(* Logix 5000 project; controller VET 1756-L62 rev 19.52; software revision 19.01; part 2 of 27 *)

        [110].S.BITS1.29   // 70-CAN-12 Falla Abrir
        [129].S.BITS1.30   // RIB-30 Falla Partida
        [129].S.BITS2.11   // RED-636-00 Enc Ext
        [36].S.BITS1.10   // 7-BIN-1060 LH
        [372].S.BITS1.8   // 110-ACD-001/1 Atollo
        [36].S.BITS1.26   // 60-VEN-002 FLL
        [119].S.BITS1.2   // 70-TDC-005 Conf. Marcha
        [141].S.BITS2.20   // 7-ROS-1140 Reset Falla
        [36].S.BITS1.27   // 60-VEN-002 FV0
        [373].S.BITS1.8   // 110-EXP-001/1 Atollo
        [46].S.BITS1.30   // 7-ROS-1069 Falla Partida
        [46].S.BITS2.7   // CON-666-00 Disable Codes
        [36].S.BITS1.28   // 60-VEN-002 FATO
        [133].S.BITS1.0   // RIB-32 Enable
        [374].S.BITS1.8   // 110-DES-001/1 Atollo
        [36].S.BITS2.7   // CON-660-00Cmd Open
        [375].S.BITS1.8   // 110-CAE-001/1 Atollo
        [141].S.BITS2.23   // 7-ROS-1140 Test
        [36].S.BITS2.20   // 60-VEN-002 Reset Falla
        [235].S.BITS1.9   // Nivel lleno Estanque Faenadora
        [36].S.BITS2.23   // 60-VEN-002 Test
        [47].S.BITS1.1   // 7-ELV-1070 Falla Resumen
        [141].S.BITS2.27   // 7-ROS-1140 Cmd. Marcha
        [47].S.BITS2.7   // CON-667-00 Disable Codes
        [129].S.BITS2.20   // RIB-30 Reset Falla
        [36].S.BITS2.27   // 60-VEN-002 Cmd. Marcha
        [141].S.BITS2.30   // 7-ROS-1140 OUT MARCHA
        [131].S.BITS1.9   // 100-TDC-001 Sobrecarga
        [48].S.BITS2.7   // CON-668-00 Disable Codes
        [110].S.BITS2.31   // 70-CAN-12 OUT OPEN
        [142].S.BITS1.7   // 70-BIN-002 LLL
        [111].S.BITS1.0   // CV-5 Enable
        [111].S.BITS1.1   // CV-5 Falla Resumen
        [87].S.BITS1.0   // TCS-28 Enable
        [46].S.BITS1.10   // 90-MMA-001 Velocidad Cero
        [87].S.BITS1.1   // TCS-28 Falla Resumen
        [156].S.BITS1.9   // 7-BIN-1155 LM
        [49].S.BITS1.10   // 90-TOR-001 Velocidad Cero
        [50].S.BITS1.8   // 90-TAB-002 Atollo
        [202].S.BITS2.11   // RED-037-00 Enc Ext
        [50].S.BITS1.10   // 90-TAB-002 Velocidad Cero
        [66].S.BITS1.4   // 60-ELV-003 Cmd. Automatico
        [442].S.BITS1.8   // 9-BIN-704 LL
        [84].S.BITS1.8   // 90-MRO-003-B Atollo
        [111].S.BITS1.2   // CV-5 Conf Pos Abrir
        [684].S.BITS2.23   // 120-CAN-070 Test
        [160].S.BITS2.27   // ROS-015-00 Cmd
        [23].S.BITS1.10   // 90-CAN-010 Conf. Abierto
        [160].S.BITS2.31   // ROS-015-00 Out
        [111].S.BITS1.4   // CV-5 Conf Pos Cerrar
        [37].S.BITS1.0   // 60-VEN-004A Enable
        [444].S.BITS1.8   // 9-BIN-706 LL
        [37].S.BITS1.26   // 60-VEN-004A FLL
        [107].S.BITS1.10   // 7-BIN-1106 LH
        [156].S.BITS1.10   // 7-BIN-1155 LH
        [37].S.BITS1.27   // 60-VEN-004A FV0
        [683].S.BITS1.8   // 120-BIN-032 LL
        [25].S.BITS1.0   // 7-CON-1025 Enable
        [143].S.BITS1.26   // 7-BBA-1142 FLL
        [156].S.BITS1.29   // M1-COMP-400 Falla Abrir
        [143].S.BITS1.27   // 7-BBA-1142 FV0
        [143].S.BITS1.28   // 7-BBA-1142 FATO
        [166].S.BITS1.2   // ROS-018-00 Run
        [49].S.BITS1.30   // 7-CON-1072 Falla Cerrar
        [683].S.BITS1.9   // 120-BIN-032 LM
        [95].S.BITS1.4   // CV-7 Conf Pos Cerrar
        [143].S.BITS1.30   // 7-BBA-1142 Falla Partida
        [95].S.BITS1.8   // 7-RED-770 LL
        [111].S.BITS1.26   // RIB-21 FLL
        [111].S.BITS1.27   // RIB-21 FV0
        [143].S.BITS2.7   // CON-684-00Cmd Open
        [95].S.BITS1.10   // 7-RED-770 LH
        [111].S.BITS1.28   // RIB-21 FATO
        [44].S.BITS1.10   // 7-TV-107X LH
        [111].S.BITS1.29   // CV-5 Falla Abrir
        [449].S.BITS1.8   // 110-VAL-001/2-1 Atollo
        [111].S.BITS1.30   // CV-5 Falla Cerrar
        [54].S.BITS1.8   // 90-ALI-002 Atollo
        [111].S.BITS2.20   // CV-5 Reset Falla
        [37].S.BITS1.28   // 60-VEN-004A FATO
        [129].S.BITS2.23   // RIB-30 Test
        [147].S.BITS1.30   // 7-CON-1146 Falla Cerrar
        [299].S.BITS1.8   // 100-TDP-006 Atollo
        [111].S.BITS2.23   // CV-5 Test
        [95].S.BITS1.26   // RIB-13 FLL
        [37].S.BITS2.7   // CON-661-00Cmd Open
        [111].S.BITS2.27   // CV-5 Cmd. Open
        [37].S.BITS2.23   // 60-VEN-004A Test
        [111].S.BITS2.30   // CV-5 OUT CLOSE
        [173].S.BITS1.28   // 70-TOR-017 FATO
        [173].S.BITS1.30   // 70-TOR-017 Falla Partida
        [173].S.BITS2.20   // 70-TOR-017 Reset Falla
        [173].S.BITS2.23   // 70-TOR-017 Test
        [173].S.BITS2.27   // 70-TOR-017 Cmd. Marcha
        [38].S.BITS1.0   // 60-TOR-002Enable
        [111].S.BITS2.31   // CV-5 OUT OPEN
        [173].S.BITS2.30   // 70-TOR-017 OUT MARCHA
        [38].S.BITS1.1   // 60-TOR-002Falla Resumen
        [143].S.BITS2.30   // 7-BBA-1142 OUT MARCHA
        [174].S.BITS1.2   // ROS-022-00 Run
        [38].S.BITS1.7   // 60-tol LLL
        [129].S.BITS2.27   // RIB-30 Cmd. Marcha
        [161].S.BITS1.0   // 7-ROS-1160 Enable
        [147].S.BITS2.7   // CON-639-00 Disable Codes
        [49].S.BITS2.7   // CON-669-00 Disable Codes
        [451].S.BITS1.8   // 110-ENF-001/2-5 Atollo
        [174].S.BITS1.7   // 70-BIN-018 LLL
        [134].S.BITS1.9   // 7-TOL-1137 LM
        [38].S.BITS1.26   // 60-TOR-002FLL
        [104].S.BITS1.9   // 90-TDC-003 Sobrecarga
        [38].S.BITS1.27   // 60-TOR-002FV0
        [55].S.BITS1.10   // 90-FIL-002 Conf. Abierto
        [142].S.BITS1.9   // 100-TDC-003 Sobrecarga
        [38].S.BITS1.28   // 60-TOR-002FATO
        [170].S.BITS1.0   // Enable
        [185].S.BITS1.9   // TOL-025-00 LM
        [87].S.BITS1.2   // TCS-28 Conf. Marcha
        [95].S.BITS1.27   // RIB-13 FV0
        [171].S.BITS2.27   // 7-VRT-1169 Cmd. Marcha
        [50].S.BITS1.30   // 7-CON-1073 Falla Cerrar
        [166].S.BITS1.7   // 70-BIN-014 LLL
        [119].S.BITS1.4   // 70-TDC-005 Cmd. Automatico
        [87].S.BITS1.4   // TCS-28 Cmd. Automatico
        [87].S.BITS1.8   // ROS-615-00 IAto
        [171].S.BITS2.30   // 7-VRT-1169 OUT MARCHA
        [70].S.BITS1.8   // 70-TOL-001 LL
        [95].S.BITS1.28   // RIB-13 FATO
        [144].S.BITS1.7   // 70-BIN-003 LLL
        [56].S.BITS1.8   // 90-VEN-002 Atollo
        [38].S.BITS2.7   // CON-662-00Cmd Open
        [194].S.BITS1.7   // 70-TOL-006 LLL
        [119].S.BITS1.26   // 70-TDC-005 FLL
        [95].S.BITS1.29   // CV-7 Falla Abrir
        [119].S.BITS1.27   // 70-TDC-005 FV0
        [462].S.BITS1.8   // 9-BIN-724 LL
        [174].S.BITS2.11   // ROS-022-00 Enc Ext
        [174].S.BITS2.27   // ROS-022-00 Cmd
        [174].S.BITS2.31   // ROS-022-00 Out
        [38].S.BITS2.20   // 60-TOR-002Reset Falla
        [119].S.BITS1.28   // 70-TDC-005 FATO
        [97].S.BITS1.10   // 7-TOL-799 LH
        [170].S.BITS1.1   // Falla Resumen
        [464].S.BITS1.8   // 9-BIN-726 LL
        [54].S.BITS1.10   // 90-ALI-002 Velocidad Cero
        [95].S.BITS1.30   // CV-7 Falla Cerrar
        [38].S.BITS2.23   // 60-TOR-002Test
        [108].S.BITS1.10   // 90-ELV-003 Velocidad Cero
        [249].S.BITS1.4   // 70-TOL-015-M Conf Pos Cerrar
        [156].S.BITS1.30   // M1-COMP-400 Falla Cerrar
        [156].S.BITS2.11   // ROS-013-00 Enc Ext
        [95].S.BITS2.11   // RED-618-00 Enc Ext
        [129].S.BITS2.30   // RIB-30 OUT MARCHA
        [129].S.BITS2.31   // RED-636-00 Out
        [163].S.BITS1.26   // 7-ROS-1162 FLL
        [130].S.BITS1.0   // 7-ROS-1129 Enable
        [87].S.BITS1.10   // ROS-615-00 IV0
        [87].S.BITS1.26   // TCS-28 FLL
        [87].S.BITS1.27   // TCS-28 FV0
        [87].S.BITS1.28   // TCS-28 FATO
        [87].S.BITS1.30   // TCS-28 Falla Partida
        [130].S.BITS1.1   // 7-ROS-1129 Falla Resumen
        [87].S.BITS2.11   // ROS-615-00 Enc Ext
        [70].S.BITS1.9   // 70-TOL-001 LM
        [70].S.BITS2.11   // RED-680-00 Enc Ext
        [87].S.BITS2.20   // TCS-28 Reset Falla
        [87].S.BITS2.23   // TCS-28 Test
        [87].S.BITS2.27   // TCS-28 Cmd. Marcha
        [87].S.BITS2.30   // TCS-28 OUT MARCHA
        [87].S.BITS2.31   // ROS-615-00 Out
        [88].S.BITS1.2   // ROS-615-01 Run
        [88].S.BITS1.7   // 70-TOL-017 LLL
        [88].S.BITS1.8   // 7-RED-001 LL
        [88].S.BITS1.9   // 7-RED-001 LM
        [146].S.BITS1.9   // 100-TDC-004 Sobrecarga
        [130].S.BITS1.2   // 7-ROS-1129 Conf. Marcha
        [88].S.BITS1.10   // 7-RED-001 LH
        [88].S.BITS2.11   // ROS-615-01 Enc Ext
        [88].S.BITS2.27   // ROS-615-01 Cmd
        [130].S.BITS1.4   // 7-ROS-1129 Cmd. Automatico
        [71].S.BITS1.0   // 90-CAN-017 Enable
        [71].S.BITS1.1   // 90-CAN-017 Falla Resumen
        [88].S.BITS2.31   // ROS-615-01 Out
        [89].S.BITS1.0   // 70-ELV-003 Enable
        [124].S.BITS1.8   // BIN-28 LL
        [130].S.BITS1.8   // BIN-31 LL
        [89].S.BITS1.1   // 70-ELV-003 Falla Resumen
        [112].S.BITS2.11   // ESP-625-00 Enc Ext
        [89].S.BITS1.2   // 70-ELV-003 Conf. Marcha
        [130].S.BITS1.9   // BIN-31 LM
        [130].S.BITS1.10   // BIN-31 LH
        [130].S.BITS1.26   // 7-ROS-1129 FLL
        [119].S.BITS1.30   // 70-TDC-005 Falla Partida
        [57].S.BITS1.8   // 90-MMA-002 Atollo
        [89].S.BITS1.4   // 70-ELV-003 Cmd. Automatico
        [119].S.BITS2.20   // 70-TDC-005 Reset Falla
        [130].S.BITS1.27   // 7-ROS-1129 FV0
        [89].S.BITS1.9   // 7-TOL-010 LM
        [95].S.BITS2.20   // CV-7 Reset Falla
        [38].S.BITS2.27   // 60-TOR-002Cmd. Marcha
        [119].S.BITS2.23   // 70-TDC-005 Test
        [166].S.BITS1.8   // 7-BIN-1165 LL
        [175].S.BITS1.10   // 100-TOR-002 Velocidad Cero
        [59].S.BITS1.8   // 7-BIN-1081 LL
        [56].S.BITS1.10   // 90-VEN-002 Velocidad Cero
        [469].S.BITS1.8   // 110-VAL-002/2-1 Atollo
        [38].S.BITS2.30   // 60-TOR-002OUT MARCHA
        [95].S.BITS2.23   // CV-7 Test
        [147].S.BITS2.27   // 7-CON-1146 Cmd. Open
        [39].S.BITS1.0   // 60-TOR-002 Enable
        [147].S.BITS2.30   // 7-CON-1146 OUT CLOSE
        [95].S.BITS2.27   // CV-7 Cmd. Open
        [119].S.BITS2.27   // 70-TDC-005 Cmd. Marcha
        [194].S.BITS1.30   // Falla Partida
        [203].S.BITS1.30   // 70-TOR-026 Falla Partida
        [95].S.BITS2.30   // CV-7 OUT CLOSE
        [119].S.BITS2.30   // 70-TDC-005 OUT MARCHA
        [152].S.BITS1.9   // 100-TDC-005 Sobrecarga
        [194].S.BITS2.11   // RED-032-00 Enc Ext
        [39].S.BITS1.2   // 60-TOR-002 Conf. Marcha
        [166].S.BITS1.9   // 7-BIN-1165 LM
        [166].S.BITS1.10   // 7-BIN-1165 LH
        [166].S.BITS2.11   // ROS-018-00 Enc Ext
        [376].S.BITS1.8   // 110-PLT-001/1 Atollo
        [39].S.BITS1.26   // 60-TOR-002 FLL
        [157].S.BITS1.9   // 100-TDC-006 Sobrecarga
        [109].S.BITS1.10   // 7-BIN-1108 LH
        [166].S.BITS2.27   // ROS-018-00 Cmd
        [62].S.BITS1.8   // 90-ALI-003 Atollo
        [155].S.BITS1.8   // TOLMAC-1 LL
        [471].S.BITS1.8   // 110-ENF-002/2-5 Atollo
        [39].S.BITS1.27   // 60-TOR-002 FV0
        [95].S.BITS2.31   // CV-7 OUT OPEN
        [302].S.BITS1.8   // 100-BCE-003 Atollo
        [156].S.BITS2.20   // M1-COMP-400 Reset Falla
        [144].S.BITS1.8   // 70-BIN-003 LL
        [162].S.BITS1.9   // 7-BIN-1161 LM
        [167].S.BITS1.9   // 100-ACV-001 Sobrecarga
        [156].S.BITS2.23   // M1-COMP-400 Test
        [144].S.BITS1.9   // 100-CAN-006 Conf. Cerrado
        [512].S.BITS1.8   // 110-ENF-001/3-4 Atollo
        [168].S.BITS1.9   // 100-FIL-002 Sobrecarga
        [166].S.BITS2.31   // ROS-018-00 Out
        [203].S.BITS2.7   // CON-038-00 Disable Codes
        [176].S.BITS1.0   // Enable
        [148].S.BITS1.7   // 70-BIN-005 LLL
        [169].S.BITS1.9   // 100-VEN-002 Sobrecarga
        [13].S.BITS1.4   // 7-CON-1013 Conf Pos Cerrar
        [148].S.BITS1.8   // 70-BIN-005 LL
        [156].S.BITS2.27   // M1-COMP-400 Cmd. Open
        [176].S.BITS1.1   // Falla Resumen
        [176].S.BITS1.2   // Conf. Marcha
        [39].S.BITS1.28   // 60-TOR-002 FATO
        [189].S.BITS1.8   // TOL-028-00 LL
        [120].S.BITS1.2   // 7-ROS-1119 Conf. Marcha
        [106].S.BITS1.9   // 90-ELV-001 Sobrecarga
        [381].S.BITS1.8   // 110-ESC-001/1 Atollo
        [203].S.BITS2.20   // 70-TOR-026 Reset Falla
        [96].S.BITS1.2   // 90-TDC-006 Conf. Marcha
        [72].S.BITS1.8   // 90-ALI-004 Atollo
        [189].S.BITS1.9   // TOL-028-00 LM
        [514].S.BITS1.8   // 110-ENF-001/3-1 Atollo
        [134].S.BITS2.7   // CON-692-00 Disable Codes
        [155].S.BITS1.10   // 100-CAN-015 Conf. Abierto
        [322].S.BITS1.9   // 100-MIX-001-M Sobrecarga
        [14].S.BITS1.4   // 7-CON-1014 Conf Pos Cerrar
        [85].S.BITS1.8   // 90-MRO-003-C Atollo
        [130].S.BITS1.28   // 7-ROS-1129 FATO
        [130].S.BITS1.30   // 7-ROS-1129 Falla Partida
        [89].S.BITS1.10   // 7-TOL-010 LH
        [163].S.BITS1.27   // 7-ROS-1162 FV0
        [89].S.BITS1.26   // 70-ELV-003 FLL
        [365].S.BITS1.9   // 110-CAN-010/1 Sobrecarga
        [89].S.BITS1.27   // 70-ELV-003 FV0
        [120].S.BITS1.8   // BIN-26 LL
        [303].S.BITS1.9   // XY-6170 Sobrecarga
        [82].S.BITS1.8   // 90-ALI-005 Atollo
        [182].S.BITS1.7   // CV-008 LLL
        [176].S.BITS1.4   // Cmd. Automatico
        [156].S.BITS2.30   // M1-COMP-400 OUT CLOSE
        [89].S.BITS1.28   // 70-ELV-003 FATO
        [80].S.BITS2.20   // 7-RED-1093 Reset Falla
        [80].S.BITS2.23   // 7-RED-1093 Test
        [189].S.BITS1.10   // TOL-028-00 LH
        [163].S.BITS1.28   // 7-ROS-1162 FATO
        [163].S.BITS1.30   // 7-ROS-1162 Falla Partida
        [172].S.BITS1.9   // 100-TOR-001 Sobrecarga
        [51].S.BITS1.2   // 7-CON-1074 Conf Pos Abrir
        [71].S.BITS1.4   // 90-CAN-017 Conf Pos Cerrar
        [519].S.BITS1.8   // 110-VAL-001/3-1 Atollo
        [92].S.BITS1.8   // 7-TOL-797 LL
        [370].S.BITS1.9   // 110-TOR-001/1 Sobrecarga
        [89].S.BITS1.30   // 70-ELV-003 Falla Partida
        [52].S.BITS1.30   // 7-CON-1075 Falla Cerrar
        [39].S.BITS2.7   // CON-663-00Cmd Open
        [39].S.BITS2.20   // 60-TOR-002 Reset Falla
        [120].S.BITS1.9   // BIN-26 LM
        [521].S.BITS1.8   // 110-ENF-001/3-5 Atollo
        [130].S.BITS2.7   // CON-637-00 Disable Codes
        [532].S.BITS1.8   // 110-ENF-002/3-4 Atollo
        [170].S.BITS1.2   // Conf. Marcha
        [170].S.BITS1.4   // Cmd. Automatico
        [170].S.BITS1.7   // 70-BIN-016 LLL
        [170].S.BITS1.8   // 7-TOL-1168 LL
        [71].S.BITS1.8   // 7-BIN-1087 LL
        [71].S.BITS1.10   // 7-BIN-1087 LH
        [71].S.BITS1.26   // 70-TDC-013 FLL
        [53].S.BITS1.2   // 7-RED-1076 Conf. Marcha
        [16].S.BITS1.4   // 7-LMG-1016 Cmd. Automatico
        [39].S.BITS2.23   // 60-TOR-002 Test
        [89].S.BITS2.7   // COM-614-01 Disable Codes
        [93].S.BITS1.8   // 90-FIL-003 Atollo
        [163].S.BITS2.30   // 7-ROS-1162 OUT MARCHA
        [89].S.BITS2.20   // 70-ELV-003 Reset Falla
        [53].S.BITS2.20   // 7-RED-1076 Reset Falla
        [71].S.BITS1.27   // 70-TDC-013 FV0
        [534].S.BITS1.8   // 110-ENF-002/3-1 Atollo
        [125].S.BITS1.0   // 70-CAN-28 Enable
        [148].S.BITS1.26   // RIB-39 FLL
        [120].S.BITS1.10   // BIN-26 LH
        [120].S.BITS1.29   // 70-CAN-39 Falla Abrir
        [17].S.BITS1.4   // 7-ELV-1017 Cmd. Automatico
        [123].S.BITS1.10   // 7-BIN-1122 LH
        [124].S.BITS1.10   // 100-CAN-019 Conf. Abierto
        [96].S.BITS1.29   // 70-CAN-23 Falla Abrir
        [148].S.BITS1.27   // RIB-39 FV0
        [203].S.BITS2.27   // 70-TOR-026 Cmd. Marcha
        [148].S.BITS1.28   // RIB-39 FATO
        [125].S.BITS1.1   // 70-CAN-28 Falla Resumen
        [107].S.BITS1.9   // 7-BIN-1106 LM
        [26].S.BITS1.4   // 7-CON-1026 Conf Pos Cerrar
        [130].S.BITS2.20   // 7-ROS-1129 Reset Falla
        [203].S.BITS2.30   // 70-TOR-026 OUT MARCHA
        [204].S.BITS2.7   // CON-039-00 Disable Codes
        [175].S.BITS1.9   // 100-TOR-002 Sobrecarga
        [304].S.BITS1.8   // 100-BCE-005 Atollo
        [54].S.BITS2.20   // 7-CON-1077 Reset Falla
        [167].S.BITS1.8   // 100-ACV-001 Atollo
        [125].S.BITS1.2   // 70-CAN-28 Conf Pos Abrir
        [96].S.BITS2.11   // RED-631-00 Enc Ext
        [305].S.BITS1.9   // 8-TOL-608 LM
        [155].S.BITS1.26   // 70-TOR-008 FLL
        [125].S.BITS1.4   // 70-CAN-28 Conf Pos Cerrar
        [31].S.BITS1.2   // 7-RED-1052 Conf. Marcha
        [112].S.BITS1.8   // 100-FIL-001 Atollo
        [108].S.BITS1.9   // 90-ELV-003 Sobrecarga
        [125].S.BITS1.8   // 7-BIN-1124 LL
        [125].S.BITS1.10   // 7-BIN-1124 LH
        [120].S.BITS2.31   // 70-CAN-39 OUT OPEN
        [167].S.BITS1.10   // 100-ACV-001 Velocidad Cero
        [125].S.BITS1.26   // RIB-28 FLL
        [206].S.BITS2.11   // LBN-040-01 Enc Ext
        [149].S.BITS1.0   // 7-CON-1148 Enable
        [209].S.BITS1.1   // 70-TOR-027 Falla Resumen
        [306].S.BITS1.9   // XY-6121 Sobrecarga
        [308].S.BITS1.8   // 100-BCE-002 Atollo
        [209].S.BITS1.2   // 70-TOR-027 Conf. Marcha
        [121].S.BITS1.0   // 70-CAN-14 Enable
        [31].S.BITS2.20   // 7-RED-1052 Reset Falla
        [149].S.BITS1.1   // 7-CON-1148 Falla Resumen
        [96].S.BITS2.31   // 90-TDC-006 OUT MARCHA
        [209].S.BITS1.4   // 70-TOR-027 Cmd. Automatico
        [125].S.BITS1.27   // RIB-28 FV0
        [121].S.BITS1.1   // 70-CAN-14 Falla Resumen
        [96].S.BITS1.8   // 7-TOL-798 LL
        [31].S.BITS2.27   // 7-RED-1052 Cmd. Marcha
        [155].S.BITS1.27   // 70-TOR-008 FV0
        [125].S.BITS1.28   // RIB-28 FATO
        [190].S.BITS1.2   // CON-029-00 Open
        [155].S.BITS1.28   // 70-TOR-008 FATO
        [539].S.BITS1.8   // 110-VEN-002/3-1 Atollo
        [125].S.BITS1.29   // 70-CAN-28 Falla Abrir
        [190].S.BITS1.4   // CON-029-00 Close
        [64].S.BITS2.11   // RED-664-00 Enc Ext
        [155].S.BITS1.30   // 100-CAN-015 Falla Cerrar
        [178].S.BITS1.9   // 7-DOS-1170-03 LM
        [130].S.BITS2.23   // 7-ROS-1129 Test
        [39].S.BITS2.27   // 60-TOR-002 Cmd. Marcha
        [190].S.BITS1.7   // 70-TOL-004 LLL
        [309].S.BITS1.9   // XY-6100 Sobrecarga
        [130].S.BITS2.27   // 7-ROS-1129 Cmd. Marcha
        [181].S.BITS1.9   // 100-TOR-004 Sobrecarga
        [113].S.BITS1.8   // 7-BIN-1112 LL
        [151].S.BITS1.9   // CON-687-00IClose
        [32].S.BITS1.4   // 7-RED-1053 Cmd. Automatico
        [109].S.BITS1.9   // 7-BIN-1108 LM
        [97].S.BITS1.26   // RIB-14 FLL
        [294].S.BITS1.29   // 80-LMG-002 Falla Pos. Izquierda
        [294].S.BITS2.26   // 80-LMG-002 Cmd. Pos . Izquierda
        [156].S.BITS2.31   // M1-COMP-400 OUT OPEN
        [192].S.BITS2.31   // CON-068-00_Out
        [121].S.BITS1.2   // 70-CAN-14 Conf Pos Abrir
        [541].S.BITS1.8   // 110-ENF-002/3-5 Atollo
        [372].S.BITS1.9   // 110-ACD-001/1 Sobrecarga
        [71].S.BITS1.28   // 70-TDC-013 FATO
        [121].S.BITS1.4   // 70-CAN-14 Conf Pos Cerrar
        [144].S.BITS2.11   // ELE-685-00 Enc Ext
        [121].S.BITS1.8   // 7-BIN-1120 LL
        [324].S.BITS1.9   // XY-6103 Conf. Cerrado
        [40].S.BITS1.0   // 7-VRT-1064 Enable
        [209].S.BITS1.30   // 70-TOR-027 Falla Partida
        [161].S.BITS1.1   // 7-ROS-1160 Falla Resumen
        [125].S.BITS1.30   // 70-CAN-28 Falla Cerrar
        [478].S.BITS1.8   // 110-TOR-004/2 Atollo
        [40].S.BITS1.2   // 7-VRT-1064 Conf. Marcha
        [57].S.BITS1.10   // 90-MMA-002 Velocidad Cero
        [176].S.BITS1.30   // Falla Partida
        [97].S.BITS1.27   // RIB-14 FV0
        [54].S.BITS2.27   // 7-CON-1077 Cmd. Open
        [191].S.BITS2.7   // CON-030-00Cmd Open
        [130].S.BITS2.30   // 7-ROS-1129 OUT MARCHA
        [71].S.BITS1.30   // 90-CAN-017 Falla Cerrar
        [97].S.BITS1.28   // RIB-14 FATO
        [130].S.BITS2.31   // OUT OPEN
        [71].S.BITS2.11   // ELE-681-00 Enc Ext
        [161].S.BITS1.2   // 7-ROS-1160 Conf. Marcha
        [495].S.BITS1.8   // 110-CAN-010/3 Atollo
        [71].S.BITS2.20   // 90-CAN-017 Reset Falla
        [40].S.BITS1.26   // 7-VRT-1064 FLL
        [71].S.BITS2.23   // 90-CAN-017 Test
        [182].S.BITS1.9   // 7-DOS-1170-05 LM
        [40].S.BITS1.27   // 7-VRT-1064 FV0
        [40].S.BITS1.28   // 7-VRT-1064 FATO
        [71].S.BITS2.27   // 90-CAN-017 Cmd. Open
        [500].S.BITS1.8   // 110-TOR-001/3 Atollo
        [55].S.BITS2.7   // CON-671-00 Disable Codes
        [40].S.BITS2.11   // RED-656-00 Enc Ext
        [40].S.BITS2.20   // 7-VRT-1064 Reset Falla
        [556].S.BITS1.9   // 120-HAR-001 Sobrecarga
        [387].S.BITS1.8   // 110-ESC-003/1 Atollo
        [98].S.BITS1.8   // 7-ELV-100 LL
        [401].S.BITS1.8   // 110-ESC-002/1 Atollo
        [121].S.BITS1.10   // 7-BIN-1120 LH
        [40].S.BITS2.23   // 7-VRT-1064 Test
        [121].S.BITS1.26   // RIB-26 FLL
        [194].S.BITS2.20   // Reset Falla
        [170].S.BITS1.9   // 7-TOL-1168 LM
        [48].S.BITS1.29   // CV-3 Falla Abrir
        [209].S.BITS2.20   // 70-TOR-027 Reset Falla
        [33].S.BITS1.4   // 7-CON-1054 Conf Pos Cerrar
        [558].S.BITS1.9   // 120-TDC-002 Sobrecarga
        [121].S.BITS1.27   // RIB-26 FV0
        [182].S.BITS1.10   // 7-DOS-1170-05 LH
        [60].S.BITS1.29   // CV-4 Falla Abrir
        [59].S.BITS1.10   // 7-BIN-1081 LH
        [71].S.BITS2.30   // 90-CAN-017 OUT CLOSE
        [55].S.BITS2.20   // 7-RED-1078 Reset Falla
        [151].S.BITS1.10   // CON-687-00IOpen
        [566].S.BITS1.9   // 120-HAR-002 Sobrecarga
        [161].S.BITS1.4   // 7-ROS-1160 Cmd. Automatico
        [161].S.BITS1.8   // TOL-004-00 LL
        [184].S.BITS1.9   // 7-DOS-1170-06 LM
        [121].S.BITS1.28   // RIB-26 FATO
        [195].S.BITS2.11   // RED-033-00 Enc Ext
        [209].S.BITS2.27   // 70-TOR-027 Cmd. Marcha
        [116].S.BITS1.8   // 100-ELV-001 Atollo
        [81].S.BITS1.0   // 7-CON-1094 Enable
        [125].S.BITS2.11   // RED-632-00 Enc Ext
        [75].S.BITS1.7   // 70-TOL-002 LLL
        [121].S.BITS1.29   // 70-CAN-14 Falla Abrir
        [170].S.BITS1.10   // 7-TOL-1168 LH
        [60].S.BITS2.20   // CV-4 Reset Falla
        [72].S.BITS1.0   // 90-ALI-004 Enable
        [121].S.BITS1.30   // 70-CAN-14 Falla Cerrar
        [113].S.BITS2.11   // VEN-625-01 Enc Ext
        [249].S.BITS1.2   // 70-TOL-015-M Conf Pos Abrir
        [121].S.BITS2.11   // RED-629-00 Enc Ext
        [200].S.BITS2.11   // ROS-035-00 Enc Ext
        [200].S.BITS2.27   // ROS-035-00 Cmd
        [149].S.BITS1.4   // 7-CON-1148 Conf Pos Cerrar
        [89].S.BITS2.23   // 70-ELV-003 Test
        [125].S.BITS2.20   // 70-CAN-28 Reset Falla
        [168].S.BITS1.7   // 70-BIN-015 LLL
        [121].S.BITS2.20   // 70-CAN-14 Reset Falla
        [81].S.BITS1.1   // 7-CON-1094 Falla Resumen
        [128].S.BITS1.10   // 100-CAN-021 Conf. Abierto
        [185].S.BITS1.10   // TOL-025-00 LH
        [35].S.BITS1.4   // 7-CON-1055 Conf Pos Cerrar
        [121].S.BITS2.23   // 70-CAN-14 Test
        [145].S.BITS1.0   // 7-BIF-1144 Enable
        [209].S.BITS2.30   // 70-TOR-027 OUT MARCHA
        [125].S.BITS2.23   // 70-CAN-28 Test
        [121].S.BITS2.27   // 70-CAN-14 Cmd. Open
        [149].S.BITS1.8   // BIN-40 LL
        [36].S.BITS1.4   // 60-VEN-002 Cmd. Automatico
        [149].S.BITS1.9   // BIN-40 LM
        [121].S.BITS2.30   // 70-CAN-14 OUT CLOSE
        [176].S.BITS2.11   // ROS-023-00 Enc Ext
        [149].S.BITS1.10   // BIN-40 LH
        [122].S.BITS1.8   // 100-TDP-001 Atollo
        [210].S.BITS2.11   // LBN-041-01 Enc Ext
        [125].S.BITS2.27   // 70-CAN-28 Cmd. Open
        [121].S.BITS2.31   // 70-CAN-14 OUT OPEN
        [568].S.BITS1.9   // 120-TDC-003 Sobrecarga
        [176].S.BITS2.20   // Reset Falla
        [576].S.BITS1.9   // 120-HAR-003 Sobrecarga
        [145].S.BITS1.1   // 7-BIF-1144 Falla Resumen
        [172].S.BITS1.7   // 70-BIN-017 LLL
        [182].S.BITS2.11   // ROS-067-00 Enc Ext
        [200].S.BITS2.31   // ROS-035-00 Out
        [170].S.BITS1.28   // FATO
        [37].S.BITS1.30   // 60-VEN-004A Falla Partida
        [176].S.BITS2.27   // Cmd. Marcha
        [176].S.BITS2.30   // OUT MARCHA
        [373].S.BITS1.9   // 110-EXP-001/1 Sobrecarga
        [197].S.BITS1.8   // BINMICROB-1 LL
        [560].S.BITS2.27   // CV-11 Cmd. Open
        [187].S.BITS2.7   // CON-027-00Cmd Open
        [197].S.BITS2.31   // MAG-034-01_Out
        [198].S.BITS1.1   // Falla Resumen
        [164].S.BITS1.7   // 70-BIN-013 LLL
        [56].S.BITS2.7   // CON-672-00 Disable Codes
        [560].S.BITS2.30   // CV-11 OUT CLOSE
        [149].S.BITS1.26   // 70-TOR-005 FLL
        [197].S.BITS1.9   // BINMICROB-1 LM
        [89].S.BITS2.27   // 70-ELV-003 Cmd. Marcha
        [194].S.BITS2.27   // Cmd. Marcha
        [164].S.BITS1.8   // 7-BIN-1163 LL
        [374].S.BITS1.9   // 110-DES-001/1 Sobrecarga
        [149].S.BITS1.27   // 70-TOR-005 FV0
        [198].S.BITS1.4   // Cmd. Automatico
        [98].S.BITS1.0   // 90-TDC-007 Enable
        [581].S.BITS1.9   // 120-TDC-005 Sobrecarga
        [132].S.BITS1.10   // 100-CAN-001 Conf. Abierto
        [155].S.BITS2.27   // 100-CAN-015 Cmd. Open
        [123].S.BITS1.26   // 70-TDC-016 FLL
        [194].S.BITS2.30   // OUT MARCHA
        [186].S.BITS1.2   // CON-026-00 Open
        [194].S.BITS2.31   // RED-032-00 Out
        [123].S.BITS1.27   // 70-TDC-016 FV0
        [81].S.BITS1.2   // 7-CON-1094 Conf Pos Abrir
        [98].S.BITS1.1   // 90-TDC-007 Falla Resumen
        [591].S.BITS1.9   // 120-TDC-006 Sobrecarga
        [123].S.BITS1.28   // 70-TDC-016 FATO
        [123].S.BITS1.30   // 100-CAN-018 Falla Cerrar
        [81].S.BITS1.4   // 7-CON-1094 Conf Pos Cerrar
        [39].S.BITS1.4   // 60-TOR-002 Cmd. Automatico
        [149].S.BITS1.28   // 70-TOR-005 FATO
        [601].S.BITS1.9   // 120-TDC-007 Sobrecarga
        [611].S.BITS1.9   // 120-TDC-008 Sobrecarga
        [168].S.BITS2.11   // ROS-019-00 Enc Ext
        [89].S.BITS2.30   // 70-ELV-003 OUT MARCHA
        [72].S.BITS1.1   // 90-ALI-004 Falla Resumen
        [135].S.BITS1.10   // 100-CAN-002 Conf. Abierto
        [98].S.BITS1.2   // 90-TDC-007 Conf. Marcha
        [131].S.BITS1.2   // 100-TDC-001 Conf. Marcha
        [570].S.BITS2.27   // CV-12 Cmd. Open
        [123].S.BITS2.27   // 100-CAN-018 Cmd. Open
        [123].S.BITS2.30   // 100-CAN-018 OUT CLOSE
        [161].S.BITS1.9   // TOL-004-00 LM
        [40].S.BITS1.4   // 7-VRT-1064 Cmd. Automatico
        [62].S.BITS1.10   // 90-ALI-003 Velocidad Cero
        [149].S.BITS1.30   // 7-CON-1148 Falla Cerrar
        [89].S.BITS2.31   // COM-614-01_Out
        [90].S.BITS1.0   // 70-TDC-018 Enable
        [41].S.BITS1.2   // 7-MMA-1065 Conf. Marcha
        [570].S.BITS2.30   // CV-12 OUT CLOSE
        [57].S.BITS1.30   // 7-CON-1080 Falla Cerrar
        [90].S.BITS1.1   // 70-TDC-018 Falla Resumen
        [90].S.BITS1.2   // 70-TDC-018 Conf. Marcha
        [164].S.BITS1.26   // FLL
        [90].S.BITS1.4   // 70-TDC-018 Cmd. Automatico
        [98].S.BITS1.4   // 90-TDC-007 Cmd. Automatico
        [164].S.BITS1.27   // FV0
        [72].S.BITS1.4   // 90-ALI-004 Cmd. Automatico
        [40].S.BITS2.27   // 7-VRT-1064 Cmd. Marcha
        [678].S.BITS2.27   // 120-CAN-067 Cmd. Open
        [57].S.BITS2.7   // CON-673-00 Disable Codes
        [680].S.BITS2.27   // 120-CAN-068 Cmd. Open
        [187].S.BITS1.9   // 100-TOR-006 Sobrecarga
        [58].S.BITS2.7   // CON-674-00 Disable Codes
        [41].S.BITS1.0   // 7-MMA-1065 Enable
        [201].S.BITS1.26   // 70-TOR-025 FLL
        [201].S.BITS1.27   // 70-TOR-025 FV0
        [201].S.BITS1.28   // 70-TOR-025 FATO
        [201].S.BITS1.30   // 7-DOS-1170a Falla Cerrar
        [201].S.BITS2.11   // ELE-036-00 Enc Ext
        [125].S.BITS2.30   // 70-CAN-28 OUT CLOSE
        [98].S.BITS1.26   // 90-TDC-007 FLL
        [98].S.BITS1.27   // 90-TDC-007 FV0
        [191].S.BITS2.31   // CON-030-00_Out
        [193].S.BITS1.9   // 100-TOR-007 Sobrecarga
        [98].S.BITS1.28   // 90-TDC-007 FATO
        [58].S.BITS2.20   // 60-MRO-001-a Reset Falla
        [41].S.BITS1.26   // 7-MMA-1065 FLL
        [145].S.BITS1.8   // BIN-38 LL
        [161].S.BITS1.10   // TOL-004-00 LH
        [81].S.BITS1.26   // RIB-06 FLL
        [72].S.BITS1.26   // 90-ALI-004 FLL
        [72].S.BITS1.27   // 90-ALI-004 FV0
        [72].S.BITS1.28   // 90-ALI-004 FATO
        [72].S.BITS1.30   // 90-ALI-004 Falla Partida
        [81].S.BITS1.27   // RIB-06 FV0
        [98].S.BITS1.30   // 90-TDC-007 Falla Partida
        [81].S.BITS1.28   // RIB-06 FATO
        [41].S.BITS2.20   // 7-MMA-1065 Reset Falla
        [41].S.BITS1.27   // 7-MMA-1065 FV0
        [186].S.BITS1.4   // CON-026-00 Close
        [145].S.BITS1.9   // BIN-38 LM
        [192].S.BITS1.2   // CON-068-00 Open
        [145].S.BITS1.10   // BIN-38 LH
        [58].S.BITS2.27   // 60-MRO-001-a Cmd. Marcha
        [98].S.BITS2.20   // 90-TDC-007 Reset Falla
        [190].S.BITS2.7   // CON-029-00Cmd Open
        [145].S.BITS1.26   // 70-TOR-003 FLL
        [59].S.BITS2.7   // CON-675-00 Disable Codes
        [41].S.BITS1.28   // 7-MMA-1065 FATO
        [41].S.BITS2.23   // 7-MMA-1065 Test
        [42].S.BITS1.0   // 7-FLT-1066 Enable
        [90].S.BITS1.26   // 70-TDC-018 FLL
        [90].S.BITS1.27   // 70-TDC-018 FV0
        [42].S.BITS1.29   // 90-CAN-013 Falla Abrir
        [42].S.BITS2.20   // 7-FLT-1066 Reset Falla
        [72].S.BITS2.11   // RED-682-00 Enc Ext
        [42].S.BITS2.23   // 7-FLT-1066 Test
        [192].S.BITS1.4   // CON-068-00 Close
        [145].S.BITS1.27   // 70-TOR-003 FV0
        [114].S.BITS1.2   // 7-ROS-1113 Conf. Marcha
        [43].S.BITS1.0   // 7-VEN-1067 Enable
        [145].S.BITS1.28   // 70-TOR-003 FATO
        [90].S.BITS1.28   // 70-TDC-018 FATO
        [72].S.BITS2.20   // 90-ALI-004 Reset Falla
        [72].S.BITS2.23   // 90-ALI-004 Test
        [161].S.BITS1.26   // 7-ROS-1160 FLL
        [161].S.BITS1.27   // 7-ROS-1160 FV0
        [43].S.BITS1.2   // 7-VEN-1067 Conf. Marcha
        [145].S.BITS2.11   // RED-686-00 Enc Ext
        [176].S.BITS2.31   // ROS-023-00 Out
        [161].S.BITS1.28   // 7-ROS-1160 FATO
        [190].S.BITS2.27   // CON-029-00 Disable Codes
        [43].S.BITS1.26   // 7-VEN-1067 FLL
        [43].S.BITS1.27   // 7-VEN-1067 FV0
        [145].S.BITS2.20   // 7-BIF-1144 Reset Falla
        [145].S.BITS2.23   // 7-BIF-1144 Test
        [43].S.BITS1.28   // 7-VEN-1067 FATO
        [192].S.BITS1.7   // 70-TOL-005 LLL
        [43].S.BITS2.20   // 7-VEN-1067 Reset Falla
        [72].S.BITS2.27   // 90-ALI-004 Cmd. Marcha
        [203].S.BITS1.0   // 70-TOR-026 Enable
        [161].S.BITS1.30   // 7-ROS-1160 Falla Partida
        [90].S.BITS1.30   // 70-TDC-018 Falla Partida
        [125].S.BITS2.31   // 70-CAN-28 OUT OPEN
        [43].S.BITS2.23   // 7-VEN-1067 Test
        [375].S.BITS1.9   // 110-CAE-001/1 Sobrecarga
        [161].S.BITS2.20   // 7-ROS-1160 Reset Falla
        [65].S.BITS2.11   // RED-670-00 Enc Ext
        [72].S.BITS2.30   // 90-ALI-004 OUT MARCHA
        [151].S.BITS1.26   // 70-TOR-006 FLL
        [196].S.BITS1.9   // 7-DOS-1170-12 LM
        [90].S.BITS2.7   // CON-616-00Cmd Open
        [188].S.BITS1.1   // Falla Resumen
        [407].S.BITS1.8   // 110-ESC-004/1 Atollo
        [43].S.BITS2.27   // 7-VEN-1067 Cmd. Marcha
        [114].S.BITS1.29   // 70-CAN-25 Falla Abrir
        [376].S.BITS1.9   // 110-PLT-001/1 Sobrecarga
        [98].S.BITS2.23   // 90-TDC-007 Test
        [190].S.BITS2.31   // CON-029-00_Out
        [149].S.BITS2.20   // 7-CON-1148 Reset Falla
        [44].S.BITS1.0   // 90-FIL-001 Enable
        [381].S.BITS1.9   // 110-ESC-001/1 Sobrecarga
        [98].S.BITS2.27   // 90-TDC-007 Cmd. Marcha
        [170].S.BITS1.30   // Falla Partida
        [199].S.BITS1.9   // 100-TOR-009 Sobrecarga
        [312].S.BITS1.8   // 100-BCE-001 Atollo
        [202].S.BITS1.9   // 100-TOR-010 Sobrecarga
        [682].S.BITS2.27   // 120-CAN-069 Cmd. Open
        [66].S.BITS1.30   // 60-ELV-003 Falla Partida
        [197].S.BITS1.10   // BINMICROB-1 LH
        [68].S.BITS1.8   // RED-678-00 IAto
        [90].S.BITS2.20   // 70-TDC-018 Reset Falla
        [81].S.BITS1.29   // 7-CON-1094 Falla Abrir
        [81].S.BITS1.30   // 7-CON-1094 Falla Cerrar
        [151].S.BITS1.27   // 70-TOR-006 FV0
        [151].S.BITS1.28   // 70-TOR-006 FATO
        [146].S.BITS1.7   // 70-BIN-004 LLL
        [72].S.BITS1.10   // 90-ALI-004 Velocidad Cero
        [114].S.BITS2.31   // 70-CAN-25 OUT OPEN
        [98].S.BITS2.30   // 90-TDC-007 OUT MARCHA
        [68].S.BITS1.10   // RED-678-00 IV0
        [90].S.BITS2.23   // 70-TDC-018 Test
        [205].S.BITS1.9   // 100-TOR-036 Sobrecarga
        [44].S.BITS1.26   // 60-MMA-001 FLL
        [161].S.BITS2.23   // 7-ROS-1160 Test
        [44].S.BITS1.27   // 60-MMA-001 FV0
        [387].S.BITS1.9   // 110-ESC-003/1 Sobrecarga
        [44].S.BITS1.28   // 60-MMA-001 FATO
        [44].S.BITS2.7   // CON-665-01Cmd Open
        [44].S.BITS2.20   // 90-FIL-001 Reset Falla
        [99].S.BITS1.0   // 70-CAN-33 Enable
        [99].S.BITS1.1   // 70-CAN-33 Falla Resumen
        [99].S.BITS1.2   // 70-CAN-33 Conf Pos Abrir
        [99].S.BITS1.4   // 70-CAN-33 Conf Pos Cerrar
        [99].S.BITS1.8   // TOLVIR-MRO1 LL
        [99].S.BITS1.10   // TOLVIR-MRO1 LH
        [99].S.BITS1.26   // RIB-15 FLL
        [99].S.BITS1.27   // RIB-15 FV0
        [99].S.BITS1.28   // RIB-15 FATO
        [99].S.BITS1.29   // 70-CAN-33 Falla Abrir
        [99].S.BITS1.30   // 70-CAN-33 Falla Cerrar
        [99].S.BITS2.11   // ESP-619-00 Enc Ext
        [99].S.BITS2.20   // 70-CAN-33 Reset Falla
        [99].S.BITS2.23   // 70-CAN-33 Test
        [99].S.BITS2.27   // 70-CAN-33 Cmd. Open
        [99].S.BITS2.30   // 70-CAN-33 OUT CLOSE
        [99].S.BITS2.31   // 70-CAN-33 OUT OPEN
        [100].S.BITS1.0   // 70-CAN-34 Enable
        [73].S.BITS2.7   // CON-683-00 Disable Codes
        [44].S.BITS2.23   // 90-FIL-001 Test
        [44].S.BITS2.27   // 90-FIL-001 Cmd. Open
        [44].S.BITS2.30   // 90-FIL-001 OUT CLOSE
        [186].S.BITS2.7   // CON-026-00Cmd Open
        [100].S.BITS1.1   // 70-CAN-34 Falla Resumen
        [100].S.BITS1.2   // 70-CAN-34 Conf Pos Abrir
        [100].S.BITS1.4   // 70-CAN-34 Conf Pos Cerrar
        [100].S.BITS1.29   // 70-CAN-34 Falla Abrir
        [100].S.BITS1.30   // 70-CAN-34 Falla Cerrar
        [100].S.BITS2.11   // VEN-619-01 Enc Ext
        [100].S.BITS2.20   // 70-CAN-34 Reset Falla
        [100].S.BITS2.23   // 70-CAN-34 Test
        [100].S.BITS2.27   // 70-CAN-34 Cmd. Open
        [100].S.BITS2.30   // 70-CAN-34 OUT CLOSE
        [100].S.BITS2.31   // 70-CAN-34 OUT OPEN
        [101]   // 70-BIF-003
        [101].S.BITS1.0   // 70-BIF-003 Enable
        [101].S.BITS1.1   // 70-BIF-003 Falla Resumen
        [101].S.BITS1.4   // 70-BIF-003 Conf. Pos. Derecha
        [101].S.BITS1.26   // RIB-16 FLL
        [101].S.BITS1.27   // RIB-16 FV0
        [101].S.BITS1.28   // RIB-16 FATO
        [101].S.BITS1.30   // 70-BIF-003 Falla Pos. Derecha
        [101].S.BITS2.20   // 70-BIF-003 Reset Falla
        [101].S.BITS2.23   // 70-BIF-003 Test
        [101].S.BITS2.27   // 70-BIF-003 Cmd. Pos. Derecha
        [101].S.BITS2.30   // 70-BIF-003 Out Izquierda
        [101].S.BITS2.31   // 70-BIF-003 Out Derecha
        [102].S.BITS2.11   // ROS-621-00 Enc Ext
        [103].S.BITS1.0   // 90-VEN-004 Enable
        [103].S.BITS1.1   // 90-VEN-004 Falla Resumen
        [103].S.BITS1.2   // 90-VEN-004 Conf. Marcha
        [103].S.BITS1.4   // 90-VEN-004 Cmd. Automatico
        [103].S.BITS1.26   // 90-VEN-004 FLL
        [103].S.BITS1.27   // 90-VEN-004 FV0
        [103].S.BITS1.28   // 90-VEN-004 FATO
        [103].S.BITS1.30   // 90-VEN-004 Falla Partida
        [103].S.BITS2.11   // ROS-621-01 Enc Ext
        [103].S.BITS2.20   // 90-VEN-004 Reset Falla
        [103].S.BITS2.23   // 90-VEN-004 Test
        [103].S.BITS2.27   // 90-VEN-004 Cmd. Marcha
        [103].S.BITS2.30   // 90-VEN-004 OUT MARCHA
        [103].S.BITS2.31   // 90-VEN-004 OUT MARCHA
        [684].S.BITS2.27   // 120-CAN-070 Cmd. Open
        [208].S.BITS1.9   // 100-TOR-012 Sobrecarga
        [25].S.BITS1.1   // 7-CON-1025 Falla Resumen
        [42].S.BITS1.4   // 7-FLT-1066 Cmd. Automatico
        [45].S.BITS1.0   // 7-ROS-1068 Enable
        [126].S.BITS1.8   // 100-TDP-002 Atollo
        [161].S.BITS2.27   // 7-ROS-1160 Cmd. Marcha
        [131].S.BITS1.29   // 70-CAN-24 Falla Abrir
        [43].S.BITS1.4   // 7-VEN-1067 Cmd. Automatico
        [502].S.BITS1.8   // 110-ACD-001/3 Atollo
        [211].S.BITS1.9   // 100-TOR-013 Sobrecarga
        [45].S.BITS1.10   // 90-VEN-001 Velocidad Cero
        [186].S.BITS2.27   // CON-026-00 Disable Codes
        [151].S.BITS1.30   // 7-CON-1151 Falla Cerrar
        [82].S.BITS1.10   // 90-ALI-005 Velocidad Cero
        [115].S.BITS1.2   // 100-TOR-022 Conf. Marcha
        [92].S.BITS1.10   // 7-TOL-797 LH
        [115].S.BITS1.8   // 7-BIN-1114 LL
        [115].S.BITS1.10   // 7-BIN-1114 LH
        [68].S.BITS1.29   // 70-FIL-001 Falla Abrir
        [115].S.BITS1.29   // 70-CAN-37 Falla Abrir
        [126].S.BITS1.10   // 100-TDP-002 Velocidad Cero
        [503].S.BITS1.8   // 110-EXP-001/3 Atollo
        [68].S.BITS2.11   // RED-678-00 Enc Ext
        [203].S.BITS1.4   // 70-TOR-026 Cmd. Automatico
        [45].S.BITS1.29   // 60-FIL-001 Falla Abrir
        [44].S.BITS1.4   // 90-FIL-001 Conf Pos Cerrar
        [81].S.BITS2.7   // CON-612-00 Disable Codes
        [146].S.BITS2.7   // CON-638-00 Disable Codes
        [25].S.BITS1.29   // 7-CON-1025 Falla Abrir
        [313].S.BITS1.9   // XY-6102 Sobrecarga
        [126].S.BITS2.11   // RED-633-00 Enc Ext
        [414].S.BITS1.8   // 110-TOR-002/1 Atollo
        [131].S.BITS1.8   // 100-TDC-001 Atollo
        [81].S.BITS2.20   // 7-CON-1094 Reset Falla
        [104].S.BITS1.29   // 70-CAN-19 Falla Abrir
        [25].S.BITS1.30   // 7-CON-1025 Falla Cerrar
        [45].S.BITS2.20   // 7-ROS-1068 Reset Falla
        [323].S.BITS1.8   // 100-VIB-001 Atollo
        [66].S.BITS1.0   // 60-ELV-003 Enable
        [66].S.BITS1.1   // 60-ELV-003 Falla Resumen
        [45].S.BITS2.23   // 7-ROS-1068 Test
        [415].S.BITS1.8   // 110-TOR-003/1 Atollo
        [66].S.BITS1.2   // 60-ELV-003 Conf. Marcha
        [25].S.BITS2.20   // 7-CON-1025 Reset Falla
        [66].S.BITS1.8   // RED-676-00 IAto
        [66].S.BITS1.10   // RED-676-00 IV0
        [416].S.BITS1.8   // 110-ELV-002/1 Atollo
        [214].S.BITS1.9   // 7-ETQ-1179a LM
        [66].S.BITS1.26   // 60-ELV-003 FLL
        [45].S.BITS2.31   // 90-VEN-001 OUT MARCHA
        [46].S.BITS1.0   // 7-ROS-1069 Enable
        [104].S.BITS2.7   // COM-620-01 Disable Codes
        [115].S.BITS2.11   // ROS-627-00 Enc Ext
        [134].S.BITS1.8   // 7-TOL-1137 LL
        [46].S.BITS1.2   // 7-ROS-1069 Conf. Marcha
        [217].S.BITS1.9   // 7-ETQ-1179b LM
        [218].S.BITS1.9   // 100-TOR-038 Sobrecarga
        [504].S.BITS1.8   // 110-DES-001/3 Atollo
        [90].S.BITS2.27   // 70-TDC-018 Cmd. Marcha
        [45].S.BITS1.4   // 7-ROS-1068 Cmd. Automatico
        [417].S.BITS1.8   // 110-TOL-006/1 Atollo
        [418].S.BITS1.8   // 110-TOR-004/1 Atollo
        [69].S.BITS1.8   // RED-679-00 IAto
        [90].S.BITS2.30   // 70-TDC-018 OUT MARCHA
        [425].S.BITS1.8   // 110-CAN-010/2 Atollo
        [142].S.BITS1.8   // 100-TDC-003 Atollo
        [41].S.BITS1.29   // 90-CAN-012 Falla Abrir
        [46].S.BITS1.26   // 7-ROS-1069 FLL
        [46].S.BITS1.27   // 7-ROS-1069 FV0
        [430].S.BITS1.8   // 110-TOR-001/2 Atollo
        [81].S.BITS2.23   // 7-CON-1094 Test
        [46].S.BITS1.4   // 7-ROS-1069 Cmd. Automatico
        [198].S.BITS1.7   // 70-TOL-008 LLL
        [47].S.BITS1.30   // 7-ELV-1070 Falla Partida
        [93].S.BITS1.10   // 90-FIL-003 Velocidad Cero
        [66].S.BITS1.27   // 60-ELV-003 FV0
        [52].S.BITS1.29   // 7-CON-1075 Falla Abrir
        [149].S.BITS2.23   // 7-CON-1148 Test
        [53].S.BITS1.29   // 90-CAN-015 Falla Abrir
        [74].S.BITS1.2   // 7-MRO-1089b Conf. Marcha
        [116].S.BITS1.2   // 7-ROS-1115 Conf. Marcha
        [96].S.BITS1.10   // 7-TOL-798 LH
        [116].S.BITS1.29   // 70-CAN-26 Falla Abrir
        [61].S.BITS1.29   // 90-CAN-016 Falla Abrir
        [116].S.BITS2.11   // ROS-627-01 Enc Ext
        [220].S.BITS1.9   // 7-ETQ-1179c LM
        [432].S.BITS1.8   // 110-ACD-001/2 Atollo
        [433].S.BITS1.8   // 110-EXP-001/2 Atollo
        [63].S.BITS2.31   // 90-MRO-001-A OUT MARCHA
        [401].S.BITS1.9   // 110-ESC-002/1 Sobrecarga
        [98].S.BITS1.10   // 7-ELV-100 LH
        [66].S.BITS1.28   // 60-ELV-003 FATO
        [66].S.BITS2.11   // RED-676-00 Enc Ext
        [66].S.BITS2.20   // 60-ELV-003 Reset Falla
        [66].S.BITS2.23   // 60-ELV-003 Test
        [66].S.BITS2.27   // 60-ELV-003 Cmd. Marcha
        [66].S.BITS2.30   // 60-ELV-003 OUT MARCHA
        [66].S.BITS2.31   // RED-676-00 Out
        [182].S.BITS2.31   // 100-TOR-037 OUT MARCHA
        [90].S.BITS2.31   // CON-616-00_Out
        [81].S.BITS2.27   // 7-CON-1094 Cmd. Open
        [198].S.BITS1.30   // Falla Partida
        [198].S.BITS2.7   // MAG-034-02 Disable Codes
        [198].S.BITS2.31   // MAG-034-02 Cmd Der
        [81].S.BITS2.30   // 7-CON-1094 OUT CLOSE
        [91].S.BITS1.0   // CV-6 Enable
        [46].S.BITS1.28   // 7-ROS-1069 FATO
        [91].S.BITS1.1   // CV-6 Falla Resumen
        [64].S.BITS2.31   // 90-MRO-001-B OUT MARCHA
        [407].S.BITS1.9   // 110-ESC-004/1 Sobrecarga
        [65].S.BITS2.31   // 90-MRO-001-C OUT MARCHA
        [46].S.BITS2.20   // 7-ROS-1069 Reset Falla
        [60].S.BITS1.2   // CV-4 Conf Pos Abrir
        [46].S.BITS2.23   // 7-ROS-1069 Test
        [105].S.BITS1.9   // 7-BIN-1104 LM
        [46].S.BITS2.27   // 7-ROS-1069 Cmd. Marcha
        [117].S.BITS1.26   // RIB-24 FLL
        [414].S.BITS1.9   // 110-TOR-002/1 Sobrecarga
        [415].S.BITS1.9   // 110-TOR-003/1 Sobrecarga
        [71].S.BITS1.29   // 90-CAN-017 Falla Abrir
        [149].S.BITS2.27   // 7-CON-1148 Cmd. Open
        [149].S.BITS2.30   // 7-CON-1148 OUT CLOSE
        [188].S.BITS1.2   // Conf. Marcha
        [67].S.BITS1.29   // CV-TOL-001 Falla Abrir
        [117].S.BITS1.27   // RIB-24 FV0
        [155].S.BITS2.30   // 100-CAN-015 OUT CLOSE
        [151].S.BITS2.7   // CON-687-00Cmd Open
        [416].S.BITS1.9   // 110-ELV-002/1 Sobrecarga
        [123].S.BITS1.9   // 7-BIN-1122 LM
        [183].S.BITS1.7   // CV-009 LLL
        [49].S.BITS1.4   // 7-CON-1072 Conf Pos Cerrar
        [133].S.BITS1.1   // RIB-32 Falla Resumen
        [151].S.BITS2.20   // 7-CON-1151 Reset Falla
        [233].S.BITS1.0   // 7-LMG-1187 Enable
        [133].S.BITS1.2   // RIB-32 Conf. Marcha
        [186].S.BITS2.31   // CON-026-00_Out
        [73].S.BITS2.31   // 90-MRO-002-A OUT MARCHA
        [417].S.BITS1.9   // 110-TOL-006/1 Sobrecarga
        [151].S.BITS2.23   // 7-CON-1151 Test
        [201].S.BITS2.27   // 7-DOS-1170a Cmd. Open
        [418].S.BITS1.9   // 110-TOR-004/1 Sobrecarga
        [136].S.BITS1.10   // 100-CAN-003 Conf. Abierto
        [127].S.BITS1.8   // 7-BIN-1126 LL
        [234].S.BITS1.0   // 100-CAN-023 Enable
        [201].S.BITS2.30   // 7-DOS-1170a OUT CLOSE
        [124].S.BITS1.9   // 100-CAN-019 Conf. Cerrado
        [50].S.BITS1.4   // 7-CON-1073 Conf Pos Cerrar
        [69].S.BITS2.11   // RED-679-00 Enc Ext
        [51].S.BITS1.4   // 7-CON-1074 Conf Pos Cerrar
        [151].S.BITS2.27   // 7-CON-1151 Cmd. Open
        [151].S.BITS2.30   // 7-CON-1151 OUT CLOSE
        [52].S.BITS1.4   // 7-CON-1075 Conf Pos Cerrar
        [76].S.BITS1.8   // BIN-04 LL
        [425].S.BITS1.9   // 110-CAN-010/2 Sobrecarga
        [53].S.BITS1.1   // 7-RED-1076 Falla Resumen
        [46].S.BITS2.30   // 7-ROS-1069 OUT MARCHA
        [430].S.BITS1.9   // 110-TOR-001/2 Sobrecarga
        [127].S.BITS1.9   // 7-BIN-1126 LM
        [283].S.BITS1.4   // 70-MIX-001-M Cmd. Automatico
        [54].S.BITS1.1   // 7-CON-1077 Falla Resumen
        [156].S.BITS1.0   // M1-COMP-400 Enable
        [133].S.BITS1.4   // RIB-32 Cmd. Automatico
        [91].S.BITS1.2   // CV-6 Conf Pos Abrir
        [74].S.BITS2.31   // 90-MRO-002-B OUT MARCHA
        [137].S.BITS1.10   // 100-CAN-004 Conf. Abierto
        [143].S.BITS1.10   // 100-CAN-005 Conf. Abierto
        [91].S.BITS1.4   // CV-6 Conf Pos Cerrar
        [313].S.BITS2.25   // M1-TRI-095 Cmd. Pos . Izquierda
        [75].S.BITS2.31   // 90-MRO-002-C OUT MARCHA
        [133].S.BITS1.9   // 7-TOL-1134 LM
        [170].S.BITS2.11   // ROS-020-00 Enc Ext
        [161].S.BITS2.30   // 7-ROS-1160 OUT MARCHA
        [213].S.BITS1.4   // 70-TOR-029 Cmd. Automatico
        [188].S.BITS1.4   // Cmd. Automatico
        [144].S.BITS1.10   // 100-CAN-006 Conf. Abierto
        [170].S.BITS2.20   // Reset Falla
        [47].S.BITS1.0   // 7-ELV-1070 Enable
        [47].S.BITS1.9   // TV-1 LM
        [314].S.BITS1.29   // M1-BIF-096 Falla Pos. Izquierda
        [133].S.BITS1.10   // 7-TOL-1134 LH
        [170].S.BITS2.23   // Test
        [213].S.BITS1.30   // 70-TOR-029 Falla Partida
        [188].S.BITS1.7   // 70-TOL-003 LLL
        [170].S.BITS2.27   // Cmd. Marcha
        [170].S.BITS2.30   // OUT MARCHA
        [162].S.BITS1.7   // 70-BIN-012 LLL
        [164].S.BITS1.28   // FATO
        [47].S.BITS1.26   // 7-ELV-1070 FLL
        [91].S.BITS1.26   // RIB-11 FLL
        [156].S.BITS1.1   // M1-COMP-400 Falla Resumen
        [314].S.BITS2.26   // M1-BIF-096 Cmd. Pos . Izquierda
        [91].S.BITS1.27   // RIB-11 FV0
        [47].S.BITS1.27   // 7-ELV-1070 FV0
        [318].S.BITS2.26   // 76-BIF-005 Cmd. Pos . Izquierda
        [83].S.BITS2.31   // 7-CON-1096 OUT OPEN
        [133].S.BITS1.26   // RIB-32 FLL
        [170].S.BITS2.31   // ROS-020-00 Out
        [195].S.BITS2.31   // RED-033-00 Out
        [171].S.BITS1.0   // 7-VRT-1169 Enable
        [164].S.BITS2.11   // ROS-017-00 Enc Ext
        [133].S.BITS1.27   // RIB-32 FV0
        [47].S.BITS1.28   // 7-ELV-1070 FATO
        [128].S.BITS1.9   // 100-CAN-021 Conf. Cerrado
        [384].S.BITS1.29   // 8-CON-764b Falla Abrir
        [223].S.BITS1.9   // 7-TOL-1180 LM
        [133].S.BITS1.28   // RIB-32 FATO
        [171].S.BITS1.1   // 7-VRT-1169 Falla Resumen
        [188].S.BITS1.30   // Falla Partida
        [184].S.BITS1.7   // CV-010 LLL
        [196].S.BITS1.7   // 70-TOL-007 LLL
        [171].S.BITS1.2   // 7-VRT-1169 Conf. Marcha
        [133].S.BITS1.30   // RIB-32 Falla Partida
        [156].S.BITS1.2   // M1-COMP-400 Conf Pos Abrir
        [84].S.BITS2.31   // 7-CON-1097 OUT OPEN
        [384].S.BITS2.26   // L3-BIF-043 Cmd. Pos . Izquierda
        [194].S.BITS1.1   // Falla Resumen
        [133].S.BITS2.7   // CON-691-00 Disable Codes
        [171].S.BITS1.4   // 7-VRT-1169 Cmd. Automatico
        [162].S.BITS1.10   // 7-BIN-1161 LH
        [188].S.BITS2.20   // Reset Falla
        [184].S.BITS1.8   // 7-DOS-1170-06 LL
        [105].S.BITS1.29   // 70-CAN-20 Falla Abrir
        [133].S.BITS2.20   // RIB-32 Reset Falla
        [156].S.BITS1.4   // M1-COMP-400 Conf Pos Cerrar
        [132].S.BITS1.9   // 100-CAN-001 Conf. Cerrado
        [152].S.BITS1.7   // 70-BIN-007 LLL
        [117].S.BITS1.28   // RIB-24 FATO
        [203].S.BITS1.28   // 70-TOR-026 FATO
        [85].S.BITS2.31   // 90-MRO-003-C OUT MARCHA
        [91].S.BITS1.28   // RIB-11 FATO
        [239].S.BITS1.9   // 100-MMA-001 Sobrecarga
        [47].S.BITS2.23   // 7-ELV-1070 Test
        [162].S.BITS2.11   // ROS-016-00 Enc Ext
        [201].S.BITS1.8   // 100-BIN-010 LL
        [152].S.BITS1.8   // 100-TDC-005 Atollo
        [178].S.BITS2.11   // ROS-024-00 Enc Ext
        [135].S.BITS1.9   // 100-CAN-002 Conf. Cerrado
        [147].S.BITS1.10   // 100-CAN-008 Conf. Abierto
        [133].S.BITS2.23   // RIB-32 Test
        [146].S.BITS1.8   // 100-TDC-004 Atollo
        [242].S.BITS1.9   // 100-TOR-021 Sobrecarga
        [195].S.BITS1.8   // 100-BIN-008 LL
        [192].S.BITS2.7   // CON-068-00Cmd Open
        [244].S.BITS1.9   // 100-TOR-020 Sobrecarga
        [127].S.BITS1.10   // 7-BIN-1126 LH
        [47].S.BITS2.30   // 7-ELV-1070 OUT MARCHA
        [148].S.BITS1.10   // 100-CAN-009 Conf. Abierto
        [150].S.BITS1.7   // 70-BIN-006 LLL
        [150].S.BITS1.8   // 70-BIN-006 LL
        [102].S.BITS2.31   // 90-FIL-004 OUT MARCHA
        [136].S.BITS1.9   // 100-CAN-003 Conf. Cerrado
        [127].S.BITS1.26   // 70-TDC-003 FLL
        [55].S.BITS1.1   // 7-RED-1078 Falla Resumen
        [104].S.BITS2.31   // 90-TDC-003 OUT MARCHA
        [192].S.BITS2.27   // CON-068-00 Disable Codes
        [133].S.BITS2.27   // RIB-32 Cmd. Marcha
        [201].S.BITS1.10   // 100-BIN-010 LH
        [105].S.BITS2.31   // 90-TDC-004 OUT MARCHA
        [152].S.BITS2.11   // ELE-688-00 Enc Ext
        [106].S.BITS2.31   // 90-ELV-001 OUT MARCHA
        [246].S.BITS1.9   // 100-TOR-019 Sobrecarga
        [248].S.BITS1.9   // 100-TOR-018 Sobrecarga
        [152].S.BITS2.31   // 7-CON-1152 OUT OPEN
        [127].S.BITS1.27   // 70-TDC-003 FV0
        [127].S.BITS1.28   // 70-TDC-003 FATO
        [392].S.BITS2.26   // 75-BIF-003 Cmd. Pos . Izquierda
        [194].S.BITS1.2   // Conf. Marcha
        [133].S.BITS2.30   // RIB-32 OUT MARCHA
        [137].S.BITS1.9   // 100-CAN-004 Conf. Cerrado
        [188].S.BITS2.27   // Cmd. Marcha
        [143].S.BITS1.9   // 100-CAN-005 Conf. Cerrado
        [127].S.BITS1.30   // 100-CAN-020 Falla Cerrar
        [195].S.BITS1.10   // 100-BIN-008 LH
        [48].S.BITS1.7   // 60-MMA-001T LLL
        [200].S.BITS1.2   // ROS-035-00 Run
        [147].S.BITS1.8   // BIN-39 LL
        [135].S.BITS1.26   // RIB-33 FLL
        [147].S.BITS1.26   // 70-TOR-004 FLL
        [56].S.BITS1.4   // 7-CON-1079 Conf Pos Cerrar
        [133].S.BITS2.31   // CON-691-00_Out
        [70].S.BITS1.7   // 70-TOL-001 LLL
        [107].S.BITS2.31   // 90-ELV-002 OUT MARCHA
        [117].S.BITS2.7   // COM-626-01 Disable Codes
        [48].S.BITS1.8   // 60-MMA-001T LL
        [171].S.BITS1.26   // 7-VRT-1169 FLL
        [147].S.BITS1.9   // 100-CAN-008 Conf. Cerrado
        [188].S.BITS2.30   // OUT MARCHA
        [194].S.BITS1.4   // Cmd. Automatico
        [213].S.BITS1.1   // 70-TOR-029 Falla Resumen
        [127].S.BITS2.11   // RED-634-00 Enc Ext
        [434].S.BITS1.8   // 110-DES-001/2 Atollo
        [172].S.BITS2.11   // ROS-021-00 Enc Ext
        [200].S.BITS1.7   // 70-TOL-009 LLL
        [91].S.BITS1.29   // CV-6 Falla Abrir
        [108].S.BITS2.31   // 90-ELV-003 OUT MARCHA
        [91].S.BITS1.30   // CV-6 Falla Cerrar
        [57].S.BITS1.4   // 7-CON-1080 Conf Pos Cerrar
        [74].S.BITS1.29   // CV-TOL-002 Falla Abrir
        [250].S.BITS1.9   // 100-TOR-017 Sobrecarga
        [505].S.BITS1.8   // 110-CAE-001/3 Atollo
        [132]   // 70-CAN-27
        [170].S.BITS1.26   // FLL
        [170].S.BITS1.27   // FV0
        [176].S.BITS1.26   // FLL
        [176].S.BITS1.27   // FV0
        [176].S.BITS1.28   // FATO
        [176].S.BITS2.23   // Test
        [188].S.BITS1.0   // Enable
        [188].S.BITS1.26   // FLL
        [188].S.BITS1.27   // FV0
        [188].S.BITS1.28   // FATO
        [188].S.BITS2.23   // Test
        [194].S.BITS1.0   // Enable
        [194].S.BITS1.26   // FLL
        [194].S.BITS1.27   // FV0
        [194].S.BITS1.28   // FATO
        [194].S.BITS2.23   // Test
        [198].S.BITS1.0   // Enable
        [198].S.BITS1.2   // Conf. Marcha
        [198].S.BITS1.26   // FLL
        [198].S.BITS1.27   // FV0
        [198].S.BITS1.28   // FATO
        [198].S.BITS2.20   // Reset Falla
        [198].S.BITS2.23   // Test
        [198].S.BITS2.27   // Cmd. Marcha
        [198].S.BITS2.30   // OUT MARCHA
        [200].S.BITS1.8   // 7-DOS-1170 LL
        [200].S.BITS1.9   // 7-DOS-1170 LM
        [200].S.BITS1.10   // 7-DOS-1170 LH
        [202].S.BITS1.7   // 70-TOL-010 LLL
        [202].S.BITS1.10   // 100-TOR-010 Velocidad Cero
        [203].S.BITS1.8   // BINMICROB-3 LL
        [203].S.BITS1.9   // BINMICROB-3 LM
        [203].S.BITS1.10   // BINMICROB-3 LH
        [203].S.BITS1.26   // 70-TOR-026 FLL
        [203].S.BITS1.27   // 70-TOR-026 FV0
        [203].S.BITS2.23   // 70-TOR-026 Test
        [203].S.BITS2.31   // CON-038-00_Out
        [204].S.BITS1.0   // Enable
        [204].S.BITS1.1   // Falla Resumen
        [204].S.BITS1.2   // Conf. Marcha
        [204].S.BITS1.4   // Cmd. Automatico
        [204].S.BITS1.9   // 100-BIN-011 LM
        [204].S.BITS1.10   // 100-BIN-011 LH
        [204].S.BITS1.26   // FLL
        [204].S.BITS1.27   // FV0
        [204].S.BITS1.28   // FATO
        [204].S.BITS1.30   // Falla Partida
        [204].S.BITS2.20   // Reset Falla
        [204].S.BITS2.23   // Test
        [204].S.BITS2.27   // Cmd. Marcha
        [204].S.BITS2.30   // OUT MARCHA
        [204].S.BITS2.31   // CON-039-00_Out
        [205].S.BITS1.7   // LBN-040-00 LLL
        [206].S.BITS1.8   // BINMICROB-4 LL
        [206].S.BITS1.9   // BINMICROB-4 LM
        [206].S.BITS1.10   // BINMICROB-4 LH
        [206].S.BITS2.31   // LBN-040-01 Out
        [207].S.BITS1.9   // 100-BIN-012 LM
        [207].S.BITS1.10   // 100-BIN-012 LH
        [207].S.BITS2.7   // LBN-040-02Cmd Open
        [207].S.BITS2.31   // LBN-040-02_Out
        [208].S.BITS1.7   // 70-DOS-001-T LLL
        [209].S.BITS1.0   // 70-TOR-027 Enable
        [209].S.BITS1.7   // LBN-041-00 LLL
        [209].S.BITS1.8   // 7-TOL-1176 LL
        [209].S.BITS1.9   // 7-TOL-1176 LM
        [209].S.BITS1.10   // 7-TOL-1176 LH
        [209].S.BITS1.26   // 70-TOR-027 FLL
        [209].S.BITS1.27   // 70-TOR-027 FV0
        [209].S.BITS1.28   // 70-TOR-027 FATO
        [209].S.BITS2.23   // 70-TOR-027 Test
        [210].S.BITS1.0   // Enable
        [210].S.BITS1.1   // Falla Resumen
        [210].S.BITS1.2   // Conf. Marcha
        [210].S.BITS1.4   // Cmd. Automatico
        [210].S.BITS1.7   // 70-DOS-002-T LLL
        [210].S.BITS1.8   // 100-BIN-013 LL
        [210].S.BITS1.9   // 100-BIN-013 LM
        [210].S.BITS1.10   // 100-BIN-013 LH
        [210].S.BITS1.26   // FLL
        [210].S.BITS1.27   // FV0
        [210].S.BITS1.28   // FATO
        [210].S.BITS1.30   // Falla Partida
        [210].S.BITS2.20   // Reset Falla
        [210].S.BITS2.23   // Test
        [210].S.BITS2.27   // Cmd. Marcha
        [210].S.BITS2.30   // OUT MARCHA
        [210].S.BITS2.31   // LBN-041-01 Out
        [211].S.BITS1.10   // 100-TOR-013 Velocidad Cero
        [211].S.BITS2.7   // LBN-041-02Cmd Open
        [212].S.BITS1.7   // 70-DOS-003-T LLL
        [212].S.BITS1.8   // 70-DOS-003-T LL
        [212].S.BITS1.9   // 70-DOS-003-T LM
        [212].S.BITS1.10   // 70-DOS-003-T LH
        [213].S.BITS1.0   // 70-TOR-029 Enable
        [213].S.BITS1.2   // 70-TOR-029 Conf. Marcha
        [213].S.BITS1.9   // 100-BIN-014 LM
        [213].S.BITS1.10   // 100-BIN-014 LH
        [213].S.BITS1.26   // 70-TOR-029 FLL
        [213].S.BITS1.27   // 70-TOR-029 FV0
        [213].S.BITS1.28   // 70-TOR-029 FATO
        [213].S.BITS2.7   // CON-042-00Cmd Open
        [213].S.BITS2.20   // 70-TOR-029 Reset Falla
        [213].S.BITS2.23   // 70-TOR-029 Test
        [213].S.BITS2.27   // 70-TOR-029 Cmd. Marcha
        [213].S.BITS2.30   // 70-TOR-029 OUT MARCHA
        [213].S.BITS2.31   // CON-042-00_Out
        [157].S.BITS1.8   // 100-TDC-006 Atollo
        [214].S.BITS1.7   // 70-DOS-004-T LLL
        [214].S.BITS2.7   // CON-043-00Cmd Open
        [506].S.BITS1.8   // 110-PLT-001/3 Atollo
        [215].S.BITS1.8   // BINMICROB-7 LL
        [215].S.BITS1.9   // BINMICROB-7 LM
        [215].S.BITS1.10   // BINMICROB-7 LH
        [215].S.BITS2.11   // ROS-044-00 Enc Ext
        [215].S.BITS2.31   // ROS-044-00 Out
        [216].S.BITS1.7   // 70-DOS-005-T LLL
        [216].S.BITS1.8   // 100-BIN-015 LL
        [216].S.BITS1.9   // 100-BIN-015 LM
        [216].S.BITS1.10   // 100-BIN-015 LH
        [216].S.BITS2.11   // MMA-045-00 Enc Ext
        [216].S.BITS2.31   // MMA-045-00 Out
        [109].S.BITS2.31   // 90-ELV-004 OUT MARCHA
        [217].S.BITS1.10   // 7-ETQ-1179b LH
        [217].S.BITS2.11   // VEN-047-00 Enc Ext
        [112].S.BITS2.31   // 100-FIL-001 OUT MARCHA
        [113].S.BITS2.31   // 100-VEN-001 OUT MARCHA
        [252].S.BITS1.9   // 100-TOR-016 Sobrecarga
        [218].S.BITS1.7   // 70-DOS-006-T LLL
        [219].S.BITS1.8   // 100-BIN-016 LL
        [219].S.BITS1.10   // 100-BIN-016 LH
        [219].S.BITS2.11   // ROS-049-00 Enc Ext
        [219].S.BITS2.31   // ROS-049-00 Out
        [220].S.BITS1.7   // 70-DOS-007-T LLL
        [220].S.BITS1.10   // 7-ETQ-1179c LH
        [221].S.BITS1.8   // BINMICROB-9 LL
        [221].S.BITS1.9   // BINMICROB-9 LM
        [221].S.BITS1.10   // BINMICROB-9 LH
        [222].S.BITS1.7   // 70-DOS-008-T LLL
        [222].S.BITS1.8   // 100-BIN-017 LL
        [222].S.BITS1.9   // 100-BIN-017 LM
        [222].S.BITS1.10   // 100-BIN-017 LH
        [222].S.BITS2.11   // ROS-050-00 Enc Ext
        [222].S.BITS2.31   // ROS-050-00 Out
        [432].S.BITS1.9   // 110-ACD-001/2 Sobrecarga
        [115].S.BITS2.31   // 100-TOR-022 OUT MARCHA
        [153].S.BITS1.10   // 100-CAN-013 Conf. Abierto
        [223].S.BITS1.10   // 7-TOL-1180 LH
        [148].S.BITS1.9   // 100-CAN-009 Conf. Cerrado
        [223].S.BITS2.11   // MMA-051-00 Enc Ext
        [116].S.BITS2.31   // 100-ELV-001 OUT MARCHA
        [122].S.BITS2.31   // 100-TDP-001 OUT MARCHA
        [262].S.BITS1.8   // 100-DOS-001-M01 Atollo
        [224].S.BITS1.7   // 70-DOS-009-T LLL
        [224].S.BITS1.8   // 70-DOS-009-T LL
        [224].S.BITS1.9   // 70-DOS-009-T LM
        [224].S.BITS1.10   // 70-DOS-009-T LH
        [224].S.BITS2.11   // VEN-053-00 Enc Ext
        [224].S.BITS2.31   // VEN-053-00 Out
        [225].S.BITS1.0   // 7-MIX-1180 Enable
        [225].S.BITS1.1   // 7-MIX-1180 Falla Resumen
        [225].S.BITS1.2   // 7-MIX-1180 Conf. Marcha
        [225].S.BITS1.4   // 7-MIX-1180 Cmd. Automatico
        [225].S.BITS1.8   // TOL-054-00 LL
        [225].S.BITS1.9   // TOL-054-00 LM
        [225].S.BITS1.10   // IVO
        [225].S.BITS1.26   // 7-MIX-1180 FLL
        [225].S.BITS1.27   // 7-MIX-1180 FV0
        [225].S.BITS1.28   // 7-MIX-1180 FATO
        [225].S.BITS1.30   // 7-MIX-1180 Falla Partida
        [225].S.BITS2.20   // 7-MIX-1180 Reset Falla
        [225].S.BITS2.23   // 7-MIX-1180 Test
        [225].S.BITS2.27   // 7-MIX-1180 Cmd. Marcha
        [225].S.BITS2.30   // 7-MIX-1180 OUT MARCHA
        [226].S.BITS1.2   // ROS-055-00 Run
        [226].S.BITS1.7   // 70-DOS-010-T LLL
        [226].S.BITS1.8   // 70-DOS-010-T LL
        [226].S.BITS1.9   // 70-DOS-010-T LM
        [226].S.BITS1.10   // 70-DOS-010-T LH
        [226].S.BITS2.11   // ROS-055-00 Enc Ext
        [226].S.BITS2.27   // ROS-055-00 Cmd
        [226].S.BITS2.31   // ROS-055-00 Out
        [227].S.BITS1.0   // 7-RED-1181 Enable
        [227].S.BITS1.1   // 7-RED-1181 Falla Resumen
        [227].S.BITS1.2   // 7-RED-1181 Conf. Marcha
        [227].S.BITS1.4   // 7-RED-1181 Cmd. Automatico
        [227].S.BITS1.8   // BINMICROB-11 LL
        [227].S.BITS1.9   // BINMICROB-11 LM
        [227].S.BITS1.10   // BINMICROB-11 LH
        [227].S.BITS1.26   // 7-RED-1181 FLL
        [227].S.BITS1.27   // 7-RED-1181 FV0
        [227].S.BITS1.28   // 7-RED-1181 FATO
        [227].S.BITS1.30   // 7-RED-1181 Falla Partida
        [227].S.BITS2.20   // 7-RED-1181 Reset Falla
        [227].S.BITS2.23   // 7-RED-1181 Test
        [227].S.BITS2.27   // 7-RED-1181 Cmd. Marcha
        [227].S.BITS2.30   // 7-RED-1181 OUT MARCHA
        [228].S.BITS1.7   // 70-DOS-011-T LLL
        [228].S.BITS1.8   // 70-DOS-011-T LL
        [228].S.BITS1.9   // 70-DOS-011-T LM
        [228].S.BITS1.10   // 70-DOS-011-T LH
        [229].S.BITS1.0   // 7-ELV-1183 Enable
        [229].S.BITS1.1   // 7-ELV-1183 Falla Resumen
        [229].S.BITS1.2   // 7-ELV-1183 Conf. Marcha
        [229].S.BITS1.4   // 7-ELV-1183 Cmd. Automatico
        [229].S.BITS1.7   // LBN-064-00 LLL
        [229].S.BITS1.8   // LBN-064-00 LL
        [229].S.BITS1.9   // LBN-064-00 LM
        [229].S.BITS1.10   // LBN-064-00 LH
        [229].S.BITS1.26   // 7-ELV-1183 FLL
        [229].S.BITS1.27   // 7-ELV-1183 FV0
        [229].S.BITS1.28   // 7-ELV-1183 FATO
        [229].S.BITS1.30   // 7-ELV-1183 Falla Partida
        [229].S.BITS2.20   // 7-ELV-1183 Reset Falla
        [229].S.BITS2.23   // 7-ELV-1183 Test
        [229].S.BITS2.27   // 7-ELV-1183 Cmd. Marcha
        [229].S.BITS2.30   // 7-ELV-1183 OUT MARCHA
        [230].S.BITS1.7   // 70-DOS-012-T LLL
        [230].S.BITS1.8   // 70-DOS-012-T LL
        [230].S.BITS1.9   // 70-DOS-012-T LM
        [230].S.BITS1.10   // 70-DOS-012-T LH
        [231].S.BITS1.0   // 70-TOR-038 Enable
        [231].S.BITS1.1   // 70-TOR-038 Falla Resumen
        [231].S.BITS1.2   // 70-TOR-038 Conf. Marcha
        [231].S.BITS1.4   // 70-TOR-038 Cmd. Automatico
        [231].S.BITS1.26   // 70-TOR-038 FLL
        [231].S.BITS1.27   // 70-TOR-038 FV0
        [231].S.BITS1.28   // 70-TOR-038 FATO
        [231].S.BITS1.30   // 70-TOR-038 Falla Partida
        [231].S.BITS2.20   // 70-TOR-038 Reset Falla
        [231].S.BITS2.23   // 70-TOR-038 Test
        [231].S.BITS2.27   // 70-TOR-038 Cmd. Marcha
        [231].S.BITS2.30   // 70-TOR-038 OUT MARCHA
        [232].S.BITS1.7   // 70-DOS-013-T LLL
        [232].S.BITS1.8   // 100-TOL-002 LL
        [232].S.BITS1.9   // 100-TOL-002 LM
        [232].S.BITS1.10   // 100-TOL-002 LH
        [233].S.BITS1.8   // BINMICROB-13 LL
        [233].S.BITS1.9   // BINMICROB-13 LM
        [233].S.BITS1.10   // BINMICROB-13 LH
        [233].S.BITS1.26   // 70-TOR-039 FLL
        [233].S.BITS1.27   // 70-TOR-039 FV0
        [233].S.BITS1.28   // 70-TOR-039 FATO
        [233].S.BITS1.30   // 7-LMG-1187 Falla Cerrar
        [233].S.BITS2.11   // ROS-070-00 Enc Ext
        [233].S.BITS2.27   // 7-LMG-1187 Cmd. Open
        [233].S.BITS2.30   // 7-LMG-1187 OUT CLOSE
        [234].S.BITS1.7   // 70-DOS-014-T LLL
        [234].S.BITS1.8   // 7-TOL-1188 LL
        [234].S.BITS1.9   // 7-TOL-1188 LM
        [234].S.BITS1.10   // 7-TOL-1188 LH
        [234].S.BITS1.26   // FLL
        [234].S.BITS1.27   // FV0
        [234].S.BITS1.28   // FATO
        [235].S.BITS1.10   // ROS-071-00 IV0
        [235].S.BITS1.26   // 7-LRT-1189 FLL
        [235].S.BITS1.27   // 7-LRT-1189 FV0
        [235].S.BITS1.28   // 7-LRT-1189 FATO
        [235].S.BITS1.30   // 7-LRT-1189 Falla Partida
        [235].S.BITS2.11   // ROS-071-00 Enc Ext
        [235].S.BITS2.30   // 7-LRT-1189 OUT MARCHA
        [236].S.BITS1.8   // 7-TOL-1190 LL
        [236].S.BITS1.9   // 7-TOL-1190 LM
        [236].S.BITS1.10   // 7-TOL-1190 LH
        [237].S.BITS1.8   // ROS-072-00 IAto
        [237].S.BITS1.10   // ROS-072-00 IV0
        [237].S.BITS2.11   // ROS-072-00 Enc Ext
        [237].S.BITS2.31   // ROS-072-00 Out
        [238].S.BITS1.8   // TOL-073-00 LL
        [238].S.BITS1.9   // TOL-073-00 LM
        [238].S.BITS1.10   // TOL-073-00 LH
        [239].S.BITS2.11   // ROS-073-00 Enc Ext
        [240].S.BITS1.7   // 70-TOL-004/A LLL
        [240].S.BITS1.26   // FLL
        [240].S.BITS1.27   // FV0
        [240].S.BITS1.28   // FATO
        [241].S.BITS1.7   // 70-TOL-004/B LLL
        [241].S.BITS1.8   // 100-TOL-006 LL
        [241].S.BITS1.9   // 100-TOL-006 LM
        [241].S.BITS1.10   // 100-TOL-006 LH
        [241].S.BITS2.11   // ROS-074-00 Enc Ext
        [433].S.BITS1.9   // 110-EXP-001/2 Sobrecarga
        [154].S.BITS1.10   // 100-CAN-014 Conf. Abierto
        [242].S.BITS1.29   // 7-CON-1195 Falla Abrir
        [434].S.BITS1.9   // 110-DES-001/2 Sobrecarga
        [126].S.BITS2.31   // 100-TDP-002 OUT MARCHA
        [511].S.BITS1.8   // 110-ESC-001/3 Atollo
        [517].S.BITS1.8   // 110-ESC-003/3 Atollo
        [243].S.BITS1.0   // 7-CON-1196 Enable
        [243].S.BITS1.1   // 7-CON-1196 Falla Resumen
        [243].S.BITS1.2   // 7-CON-1196 Conf Pos Abrir
        [243].S.BITS1.4   // 7-CON-1196 Conf Pos Cerrar
        [243].S.BITS1.8   // 100-TOL-007 LL
        [243].S.BITS1.10   // 100-TOL-007 LH
        [243].S.BITS1.26   // FLL
        [243].S.BITS1.27   // FV0
        [243].S.BITS1.28   // FATO
        [243].S.BITS1.29   // 7-CON-1196 Falla Abrir
        [243].S.BITS1.30   // 7-CON-1196 Falla Cerrar
        [243].S.BITS2.11   // ROS-075-00 Enc Ext
        [243].S.BITS2.20   // 7-CON-1196 Reset Falla
        [243].S.BITS2.23   // 7-CON-1196 Test
        [243].S.BITS2.27   // 7-CON-1196 Cmd. Open
        [243].S.BITS2.30   // 7-CON-1196 OUT CLOSE
        [243].S.BITS2.31   // 7-CON-1196 OUT OPEN
        [244].S.BITS1.7   // 70-TOL-011 LLL
        [245].S.BITS1.0   // 7-ROS-1202 Enable
        [245].S.BITS1.1   // 7-ROS-1202 Falla Resumen
        [245].S.BITS1.2   // 7-ROS-1202 Conf. Marcha
        [245].S.BITS1.4   // 7-ROS-1202 Cmd. Automatico
        [245].S.BITS1.8   // 100-TOL-008 LL
        [245].S.BITS1.10   // 100-TOL-008 LH
        [245].S.BITS1.29   // 70-VAL-001 Falla Abrir
        [245].S.BITS2.11   // ROS-076-00 Enc Ext
        [245].S.BITS2.20   // 7-ROS-1202 Reset Falla
        [245].S.BITS2.23   // 7-ROS-1202 Test
        [245].S.BITS2.31   // 70-VAL-001 OUT OPEN
        [435].S.BITS1.9   // 110-CAE-001/2 Sobrecarga
        [131].S.BITS2.31   // 100-TDC-001 OUT MARCHA
        [158].S.BITS1.10   // 7-BIN-1157 LH
        [246].S.BITS1.10   // 100-TOR-019 Velocidad Cero
        [153].S.BITS1.9   // 100-CAN-013 Conf. Cerrado
        [134].S.BITS2.31   // 100-TDC-002 OUT MARCHA
        [142].S.BITS2.31   // 100-TDC-003 OUT MARCHA
        [264].S.BITS1.8   // 100-DOS-001-MO2 Atollo
        [247].S.BITS1.0   // COMP-A Enable
        [247].S.BITS1.1   // COMP-A Falla Resumen
        [247].S.BITS1.2   // COMP-A Conf Pos Abrir
        [247].S.BITS1.4   // COMP-A Conf Pos Cerrar
        [247].S.BITS1.8   // 7-TOL-1204 LL
        [247].S.BITS1.10   // 7-TOL-1204 LH
        [247].S.BITS1.29   // COMP-A Falla Abrir
        [247].S.BITS1.30   // COMP-A Falla Cerrar
        [247].S.BITS2.11   // ROS-077-00 Enc Ext
        [247].S.BITS2.20   // COMP-A Reset Falla
        [247].S.BITS2.23   // COMP-A Test
        [247].S.BITS2.27   // COMP-A Cmd. Open
        [247].S.BITS2.30   // COMP-A OUT CLOSE
        [247].S.BITS2.31   // COMP-A OUT OPEN
        [248].S.BITS1.7   // 70-TOL-015 LLL
        [249].S.BITS1.0   // 70-TOL-015-M Enable
        [249].S.BITS1.1   // 70-TOL-015-M Falla Resumen
        [249].S.BITS1.8   // 100-TOL-010 LL
        [249].S.BITS1.9   // 100-TOL-010 LM
        [249].S.BITS1.10   // 100-TOL-010 LH
        [249].S.BITS1.29   // 70-TOL-015-M Falla Abrir
        [249].S.BITS1.30   // 70-TOL-015-M Falla Cerrar
        [249].S.BITS2.11   // ROS-078-00 Enc Ext
        [249].S.BITS2.20   // 70-TOL-015-M Reset Falla
        [249].S.BITS2.23   // 70-TOL-015-M Test
        [249].S.BITS2.27   // 70-TOL-015-M Cmd. Open
        [249].S.BITS2.30   // 70-TOL-015-M OUT CLOSE
        [249].S.BITS2.31   // 70-TOL-015-M OUT OPEN
        [436].S.BITS1.9   // 110-PLT-001/2 Sobrecarga
        [146].S.BITS2.31   // 100-TDC-004 OUT MARCHA
        [159].S.BITS1.10   // 100-CAN-017 Conf. Abierto
        [250].S.BITS1.10   // 100-TOR-017 Velocidad Cero
        [250].S.BITS1.29   // COMP-B Falla Abrir
        [154].S.BITS1.9   // 100-CAN-014 Conf. Cerrado
        [157].S.BITS2.31   // 100-TDC-006 OUT MARCHA
        [162].S.BITS2.31   // 100-TDC-008 OUT MARCHA
        [266].S.BITS1.8   // 100-DOS-001-M03 Atollo
        [251].S.BITS1.0   // 7-ELV-004B Enable
        [251].S.BITS1.1   // 7-ELV-004B Falla Resumen
        [251].S.BITS1.2   // 7-ELV-004B Conf. Marcha
        [251].S.BITS1.4   // 7-ELV-004B Cmd. Automatico
        [251].S.BITS1.8   // 100-TOL-011 LL
        [251].S.BITS1.9   // 100-TOL-011 LM
        [251].S.BITS1.10   // 100-TOL-011 LH
        [251].S.BITS1.26   // 7-ELV-004B FLL
        [251].S.BITS1.27   // 7-ELV-004B FV0
        [251].S.BITS1.28   // 7-ELV-004B FATO
        [251].S.BITS1.30   // 7-ELV-004B Falla Partida
        [251].S.BITS2.11   // ROS-079-00 Enc Ext
        [251].S.BITS2.20   // 7-ELV-004B Reset Falla
        [251].S.BITS2.23   // 7-ELV-004B Test
        [251].S.BITS2.27   // 7-ELV-004B Cmd. Marcha
        [251].S.BITS2.30   // 7-ELV-004B OUT MARCHA
        [251].S.BITS2.31   // ROS-079-00 Out
        [441].S.BITS1.9   // 110-ESC-001/2 Sobrecarga
        [252].S.BITS1.2   // 7-RED-004C Conf. Marcha
        [163].S.BITS1.10   // 100-CAN-028 Conf. Abierto
        [252].S.BITS1.10   // 100-TOR-016 Velocidad Cero
        [252].S.BITS1.29   // 70-FIL-002 Falla Abrir
        [447].S.BITS1.9   // 110-ESC-003/2 Sobrecarga
        [167].S.BITS2.31   // 100-ACV-001 OUT MARCHA
        [520].S.BITS1.8   // 110-VEN-001/3 Atollo
        [523].S.BITS1.8   // 110-QUE-001-1 Atollo
        [253].S.BITS1.0   // 70-VAL-001B Enable
        [253].S.BITS1.1   // 70-VAL-001B Falla Resumen
        [253].S.BITS1.2   // 70-VAL-001B Conf Pos Abrir
        [253].S.BITS1.4   // 70-VAL-001B Conf Pos Cerrar
        [253].S.BITS1.8   // ROS-080-00 IAto
        [253].S.BITS1.10   // ROS-080-00 IV0
        [253].S.BITS1.26   // TDC-MIC-2 FLL
        [253].S.BITS1.27   // TDC-MIC-2 FV0
        [253].S.BITS1.28   // TDC-MIC-2 FATO
        [253].S.BITS1.29   // 70-VAL-001B Falla Abrir
        [253].S.BITS1.30   // 70-VAL-001B Falla Cerrar
        [253].S.BITS2.11   // ROS-080-00 Enc Ext
        [253].S.BITS2.20   // 70-VAL-001B Reset Falla
        [253].S.BITS2.23   // 70-VAL-001B Test
        [253].S.BITS2.27   // 70-VAL-001B Cmd. Open
        [253].S.BITS2.30   // 70-VAL-001B OUT CLOSE
        [253].S.BITS2.31   // 70-VAL-001B OUT OPEN
        [254].S.BITS1.0   // 70-BBV-001 Enable
        [254].S.BITS1.1   // 70-BBV-001 Falla Resumen
        [254].S.BITS1.2   // 70-BBV-001 Conf. Marcha
        [254].S.BITS1.4   // 70-BBV-001 Cmd. Automatico
        [254].S.BITS1.26   // 70-BBV-001 FLL
        [254].S.BITS1.27   // 70-BBV-001 FV0
        [254].S.BITS1.28   // 70-BBV-001 FATO
        [254].S.BITS1.29   // COM-VERT-1 Falla Abrir
        [254].S.BITS1.30   // 70-BBV-001 Falla Partida
        [254].S.BITS2.20   // 70-BBV-001 Reset Falla
        [254].S.BITS2.23   // 70-BBV-001 Test
        [254].S.BITS2.27   // 70-BBV-001 Cmd. Marcha
        [254].S.BITS2.30   // 70-BBV-001 OUT MARCHA
        [254].S.BITS2.31   // COM-VERT-1 OUT OPEN
        [255].S.BITS1.7   // 70-TOL-012 LLL
        [255].S.BITS1.8   // 70-TOL-012 LL
        [255].S.BITS2.11   // ROS-081-00 Enc Ext
        [256].S.BITS1.0   // 70-VAL-002 Enable
        [256].S.BITS1.1   // 70-VAL-002 Falla Resumen
        [256].S.BITS1.2   // 70-VAL-002 Conf Pos Abrir
        [256].S.BITS1.4   // 70-VAL-002 Conf Pos Cerrar
        [256].S.BITS1.29   // 70-VAL-002 Falla Abrir
        [256].S.BITS1.30   // 70-VAL-002 Falla Cerrar
        [256].S.BITS2.20   // 70-VAL-002 Reset Falla
        [256].S.BITS2.23   // 70-VAL-002 Test
        [256].S.BITS2.27   // 70-VAL-002 Cmd. Open
        [256].S.BITS2.30   // 70-VAL-002 OUT CLOSE
        [256].S.BITS2.31   // 70-VAL-002 OUT OPEN
        [257].S.BITS1.0   // 70-TDP-003 Enable
        [257].S.BITS1.1   // 70-TDP-003 Falla Resumen
        [257].S.BITS1.2   // 70-TDP-003 Conf. Marcha
        [257].S.BITS1.4   // 70-TDP-003 Cmd. Automatico
        [257].S.BITS1.26   // 70-TDP-003 FLL
        [257].S.BITS1.27   // 70-TDP-003 FV0
        [257].S.BITS1.28   // 70-TDP-003 FATO
        [257].S.BITS1.30   // 70-TDP-003 Falla Partida
        [257].S.BITS2.20   // 70-TDP-003 Reset Falla
        [257].S.BITS2.23   // 70-TDP-003 Test
        [257].S.BITS2.27   // 70-TDP-003 Cmd. Marcha
        [257].S.BITS2.30   // 70-TDP-003 OUT MARCHA
        [259].S.BITS1.0   // Enable
        [259].S.BITS1.1   // Falla Resumen
        [259].S.BITS1.2   // Conf Pos Abrir
        [259].S.BITS1.4   // Conf Pos Cerrar
        [259].S.BITS1.29   // Falla Abrir
        [259].S.BITS1.30   // Falla Cerrar
        [259].S.BITS2.20   // Reset Falla
        [259].S.BITS2.23   // Test
        [259].S.BITS2.27   // Cmd. Open
        [259].S.BITS2.30   // OUT CLOSE
        [259].S.BITS2.31   // OUT OPEN
        [260].S.BITS1.0   // Enable
        [260].S.BITS1.1   // Falla Resumen
        [260].S.BITS1.2   // Conf Pos Abrir
        [260].S.BITS1.4   // Conf Pos Cerrar
        [260].S.BITS1.7   // 70-TOL-ACE1 LLL
        [260].S.BITS1.8   // 70-TOL-ACE1 LL
        [260].S.BITS1.9   // 70-TOL-ACE1 LM
        [260].S.BITS1.10   // 70-TOL-ACE1 LH
        [260].S.BITS1.29   // Falla Abrir
        [260].S.BITS1.30   // Falla Cerrar
        [260].S.BITS2.20   // Reset Falla
        [260].S.BITS2.23   // Test
        [260].S.BITS2.27   // Cmd. Open
        [260].S.BITS2.30   // OUT CLOSE
        [260].S.BITS2.31   // OUT OPEN
        [261].S.BITS1.0   // 70-BCE-09 Enable
        [261].S.BITS1.1   // 70-BCE-09 Falla Resumen
        [261].S.BITS1.2   // 70-BCE-09 Conf. Marcha
        [261].S.BITS1.4   // 70-BCE-09 Cmd. Automatico
        [261].S.BITS1.26   // 70-BCE-09 FLL
        [261].S.BITS1.27   // 70-BCE-09 FV0
        [261].S.BITS1.28   // 70-BCE-09 FATO
        [261].S.BITS1.30   // 70-BCE-09 Falla Partida
        [261].S.BITS2.7   // CON-082-01Cmd Open
        [261].S.BITS2.20   // 70-BCE-09 Reset Falla
        [261].S.BITS2.23   // 70-BCE-09 Test
        [261].S.BITS2.27   // 70-BCE-09 Cmd. Marcha
        [261].S.BITS2.30   // 70-BCE-09 OUT MARCHA
        [261].S.BITS2.31   // CON-082-01_Out
        [162].S.BITS1.8   // 7-BIN-1161 LL
        [155].S.BITS1.9   // 100-CAN-015 Conf. Cerrado
        [450].S.BITS1.9   // 9-BIN-712 LM
        [63].S.BITS1.10   // 90-MRO-001-A Velocidad Cero
        [262].S.BITS1.10   // 100-DOS-001-M01 Velocidad Cero
        [262].S.BITS1.9   // 100-DOS-001-M01 Sobrecarga
        [262].S.BITS2.11   // RED-083-00 Enc Ext
        [461].S.BITS1.9   // 110-ESC-002/2 Sobrecarga
        [467].S.BITS1.9   // 110-ESC-004/2 Sobrecarga
        [168].S.BITS2.31   // 100-FIL-002 OUT MARCHA
        [263].S.BITS1.0   // VALV-ALIM-1 Enable
        [263].S.BITS1.1   // VALV-ALIM-1 Falla Resumen
        [263].S.BITS1.2   // VALV-ALIM-1 Conf Pos Abrir
        [263].S.BITS1.4   // VALV-ALIM-1 Conf Pos Cerrar
        [263].S.BITS1.29   // VALV-ALIM-1 Falla Abrir
        [263].S.BITS1.30   // VALV-ALIM-1 Falla Cerrar
        [263].S.BITS2.20   // VALV-ALIM-1 Reset Falla
        [263].S.BITS2.23   // VALV-ALIM-1 Test
        [263].S.BITS2.27   // VALV-ALIM-1 Cmd. Open
        [263].S.BITS2.30   // VALV-ALIM-1 OUT CLOSE
        [264].S.BITS1.7   // TOL-056-00 LLL
        [265].S.BITS1.0   // 70-BCE-008 Enable
        [265].S.BITS1.1   // 70-BCE-008 Falla Resumen
        [265].S.BITS1.2   // 70-BCE-008 Conf. Marcha
        [265].S.BITS1.4   // 70-BCE-008 Cmd. Automatico
        [265].S.BITS1.26   // 70-BCE-008 FLL
        [265].S.BITS1.27   // 70-BCE-008 FV0
        [265].S.BITS1.28   // 70-BCE-008 FATO
        [265].S.BITS1.29   // SLQ1- Falla Abrir
        [265].S.BITS1.30   // 70-BCE-008 Falla Partida
        [265].S.BITS2.7   // CON-057-00Cmd Open
        [265].S.BITS2.20   // 70-BCE-008 Reset Falla
        [265].S.BITS2.23   // 70-BCE-008 Test
        [265].S.BITS2.27   // 70-BCE-008 Cmd. Marcha
        [265].S.BITS2.30   // 70-BCE-008 OUT MARCHA
        [265].S.BITS2.31   // SLQ1- OUT OPEN
        [168].S.BITS1.8   // 100-FIL-002 Atollo
        [158].S.BITS1.9   // 7-BIN-1157 LM
        [470].S.BITS1.9   // 110-VEN-002/2 Sobrecarga
        [64].S.BITS1.10   // 90-MRO-001-B Velocidad Cero
        [266].S.BITS1.10   // 100-DOS-001-M03 Velocidad Cero
        [264].S.BITS1.9   // 100-DOS-001-MO2 Sobrecarga
        [474].S.BITS1.9   // 110-TOR-002/2 Sobrecarga
        [475].S.BITS1.9   // 110-TOR-003/2 Sobrecarga
        [169].S.BITS2.31   // 100-VEN-002 OUT MARCHA
        [267].S.BITS1.0   // 70-XV-7262 Enable
        [267].S.BITS1.1   // 70-XV-7262 Falla Resumen
        [267].S.BITS1.2   // 70-XV-7262 Conf Pos Abrir
        [267].S.BITS1.4   // 70-XV-7262 Conf Pos Cerrar
        [267].S.BITS1.26   // BOM-LIQ-1 FLL
        [267].S.BITS1.27   // BOM-LIQ-1 FV0
        [267].S.BITS1.28   // BOM-LIQ-1 FATO
        [267].S.BITS1.29   // 70-XV-7262 Falla Abrir
        [267].S.BITS1.30   // 70-XV-7262 Falla Cerrar
        [267].S.BITS2.11   // MIX-058-00 Enc Ext
        [267].S.BITS2.20   // 70-XV-7262 Reset Falla
        [267].S.BITS2.23   // 70-XV-7262 Test
        [267].S.BITS2.27   // 70-XV-7262 Cmd. Open
        [267].S.BITS2.30   // 70-XV-7262 OUT CLOSE
        [267].S.BITS2.31   // 70-XV-7262 OUT OPEN
        [268].S.BITS1.7   // 70-TOL-LIS1 LLL
        [269].S.BITS1.0   // 70-BCE-001 Enable
        [269].S.BITS1.1   // 70-BCE-001 Falla Resumen
        [269].S.BITS1.2   // 70-BCE-001 Conf. Marcha
        [269].S.BITS1.4   // 70-BCE-001 Cmd. Automatico
        [269].S.BITS1.26   // 70-BCE-001 FLL
        [269].S.BITS1.27   // 70-BCE-001 FV0
        [269].S.BITS1.28   // 70-BCE-001 FATO
        [269].S.BITS1.30   // 70-BCE-001 Falla Partida
        [269].S.BITS2.11   // MIX-058-01b Enc Ext
        [269].S.BITS2.20   // 70-BCE-001 Reset Falla
        [269].S.BITS2.23   // 70-BCE-001 Test
        [269].S.BITS2.27   // 70-BCE-001 Cmd. Marcha
        [269].S.BITS2.30   // 70-BCE-001 OUT MARCHA
        [269].S.BITS2.31   // MIX-058-01b Out
        [169].S.BITS1.8   // 100-VEN-002 Atollo
        [159].S.BITS1.9   // 100-CAN-017 Conf. Cerrado
        [476].S.BITS1.9   // 110-ELV-002/2 Sobrecarga
        [65].S.BITS1.10   // 7-BIN-1084 LH
        [13].S.BITS2.31   // 7-CON-1013 OUT OPEN
        [25].S.BITS2.31   // 7-CON-1025 OUT OPEN
        [270].S.BITS1.10   // 100-DOS-001-M05 Velocidad Cero
        [270].S.BITS1.29   // VALV-ALIM-2 Falla Abrir
        [266].S.BITS1.9   // 100-DOS-001-M03 Sobrecarga
        [270].S.BITS2.7   // MIX-058-01c Disable Codes
        [478].S.BITS1.9   // 110-TOR-004/2 Sobrecarga
        [495].S.BITS1.9   // 110-CAN-010/3 Sobrecarga
        [172].S.BITS2.31   // 100-TOR-001 OUT MARCHA
        [271].S.BITS1.0   // 70-XV-7259 Enable
        [271].S.BITS1.1   // 70-XV-7259 Falla Resumen
        [271].S.BITS1.2   // 70-XV-7259 Conf Pos Abrir
        [271].S.BITS1.4   // 70-XV-7259 Conf Pos Cerrar
        [271].S.BITS1.29   // 70-XV-7259 Falla Abrir
        [271].S.BITS1.30   // 70-XV-7259 Falla Cerrar
        [271].S.BITS2.11   // MIX-058-01d Enc Ext
        [271].S.BITS2.20   // 70-XV-7259 Reset Falla
        [271].S.BITS2.23   // 70-XV-7259 Test
        [271].S.BITS2.27   // 70-XV-7259 Cmd. Open
        [271].S.BITS2.30   // 70-XV-7259 OUT CLOSE
        [271].S.BITS2.31   // 70-XV-7259 OUT OPEN
        [435].S.BITS1.8   // 110-CAE-001/2 Atollo
        [524].S.BITS1.8   // 110-QUE-001-2 Atollo
        [268].S.BITS1.8   // 100-DOS-001-M04 Atollo
        [272].S.BITS1.7   // 70-TOL-COL1 LLL
        [272].S.BITS1.29   // SLQ1-2 Falla Abrir
        [436].S.BITS1.8   // 110-PLT-001/2 Atollo
        [325].S.BITS1.8   // 100-TDC-007 Atollo
        [273].S.BITS1.0   // 70-BCE-005 Enable
        [273].S.BITS1.1   // 70-BCE-005 Falla Resumen
        [273].S.BITS1.2   // 70-BCE-005 Conf. Marcha
        [273].S.BITS1.4   // 70-BCE-005 Cmd. Automatico
        [273].S.BITS1.26   // 70-BCE-005 FLL
        [273].S.BITS1.27   // 70-BCE-005 FV0
        [273].S.BITS1.28   // 70-BCE-005 FATO
        [273].S.BITS1.30   // 70-BCE-005 Falla Partida
        [273].S.BITS2.20   // 70-BCE-005 Reset Falla
        [273].S.BITS2.23   // 70-BCE-005 Test
        [273].S.BITS2.27   // 70-BCE-005 Cmd. Marcha
        [273].S.BITS2.30   // 70-BCE-005 OUT MARCHA
        [273].S.BITS2.31   // OUT MARCHA
        [172].S.BITS1.8   // 100-TOR-001 Atollo
        [163].S.BITS1.9   // 100-CAN-028 Conf. Cerrado
        [500].S.BITS1.9   // 110-TOR-001/3 Sobrecarga
        [73].S.BITS1.10   // 90-MRO-002-A Velocidad Cero
        [268].S.BITS1.9   // 100-DOS-001-M04 Sobrecarga
        [502].S.BITS1.9   // 110-ACD-001/3 Sobrecarga
        [503].S.BITS1.9   // 110-EXP-001/3 Sobrecarga
        [175].S.BITS2.31   // 100-TOR-002 OUT MARCHA
        [275].S.BITS1.0   // 70-XV-7254 Enable
        [275].S.BITS1.1   // 70-XV-7254 Falla Resumen
        [275].S.BITS1.2   // 70-XV-7254 Conf Pos Abrir
        [275].S.BITS1.4   // 70-XV-7254 Conf Pos Cerrar
        [275].S.BITS1.29   // 70-XV-7254 Falla Abrir
        [275].S.BITS1.30   // 70-XV-7254 Falla Cerrar
        [275].S.BITS2.20   // 70-XV-7254 Reset Falla
        [275].S.BITS2.23   // 70-XV-7254 Test
        [275].S.BITS2.27   // 70-XV-7254 Cmd. Open
        [275].S.BITS2.30   // 70-XV-7254 OUT CLOSE
        [275].S.BITS2.31   // 70-XV-7254 OUT OPEN
        [175].S.BITS1.8   // 100-TOR-002 Atollo
        [353].S.BITS1.9   // 110-CAN-001 Conf. Cerrado
        [504].S.BITS1.9   // 110-DES-001/3 Sobrecarga
        [74].S.BITS1.10   // 90-MRO-002-B Velocidad Cero
        [276].S.BITS1.7   // 70-TOL-ALI1 LLL
        [276].S.BITS1.10   // 100-DOS-001-M08 Velocidad Cero
        [270].S.BITS1.9   // 100-DOS-001-M05 Sobrecarga
        [505].S.BITS1.9   // 110-CAE-001/3 Sobrecarga
        [506].S.BITS1.9   // 110-PLT-001/3 Sobrecarga
        [178].S.BITS2.31   // 100-TOR-003 OUT MARCHA
        [277].S.BITS1.0   // 70-BCE-003 Enable
        [277].S.BITS1.1   // 70-BCE-003 Falla Resumen
        [277].S.BITS1.2   // 70-BCE-003 Conf. Marcha
        [277].S.BITS1.4   // 70-BCE-003 Cmd. Automatico
        [277].S.BITS1.26   // 70-BCE-003 FLL
        [277].S.BITS1.27   // 70-BCE-003 FV0
        [277].S.BITS1.28   // 70-BCE-003 FATO
        [277].S.BITS1.29   // VALV-ALIM-3 Falla Abrir
        [277].S.BITS1.30   // 70-BCE-003 Falla Partida
        [277].S.BITS2.20   // 70-BCE-003 Reset Falla
        [277].S.BITS2.23   // 70-BCE-003 Test
        [277].S.BITS2.27   // 70-BCE-003 Cmd. Marcha
        [277].S.BITS2.30   // 70-BCE-003 OUT MARCHA
        [277].S.BITS2.31   // VALV-ALIM-3 OUT OPEN
        [178].S.BITS1.8   // 7-DOS-1170-03 LL
        [354].S.BITS1.9   // 110-CAN-002 Conf. Cerrado
        [511].S.BITS1.9   // 110-ESC-001/3 Sobrecarga
        [75].S.BITS1.10   // 90-MRO-002-C Velocidad Cero
        [272].S.BITS1.9   // 100-DOS-001-M06 Sobrecarga
        [517].S.BITS1.9   // 110-ESC-003/3 Sobrecarga
        [520].S.BITS1.9   // 110-VEN-001/3 Sobrecarga
        [181].S.BITS2.31   // 100-TOR-004 OUT MARCHA
        [279].S.BITS1.0   // 70-XV-7267 Enable
        [279].S.BITS1.1   // 70-XV-7267 Falla Resumen
        [279].S.BITS1.2   // 70-XV-7267 Conf Pos Abrir
        [279].S.BITS1.4   // 70-XV-7267 Conf Pos Cerrar
        [279].S.BITS1.29   // 70-XV-7267 Falla Abrir
        [279].S.BITS1.30   // 70-XV-7267 Falla Cerrar
        [279].S.BITS2.20   // 70-XV-7267 Reset Falla
        [279].S.BITS2.23   // 70-XV-7267 Test
        [279].S.BITS2.27   // 70-XV-7267 Cmd. Open
        [279].S.BITS2.30   // 70-XV-7267 OUT CLOSE
        [279].S.BITS2.31   // 70-XV-7267 OUT OPEN
        [441].S.BITS1.8   // 110-ESC-001/2 Atollo
        [531].S.BITS1.8   // 110-ESC-002/3 Atollo
        [270].S.BITS1.8   // 100-DOS-001-M05 Atollo
        [280].S.BITS1.29   // SLQ1-3 Falla Abrir
        [447].S.BITS1.8   // 110-ESC-003/2 Atollo
        [280].S.BITS2.7   // CON-058-00Cmd Open
        [326].S.BITS1.8   // 8-ENF-640 LL
        [281].S.BITS1.7   // TOL-058-01 LLL
        [181].S.BITS1.8   // 100-TOR-004 Atollo
        [355].S.BITS1.9   // 110-CAN-003 Conf. Cerrado
        [523].S.BITS1.9   // 110-QUE-001-1 Sobrecarga
        [83].S.BITS1.10   // 90-MRO-003-A Velocidad Cero
        [282].S.BITS1.7   // 70-MIX-001-T LLL
        [282].S.BITS1.10   // 100-DOS-100-M11 Velocidad Cero
        [274].S.BITS1.9   // 100-DOS-001-M07 Sobrecarga
        [282].S.BITS2.11   // RED-059-00 Enc Ext
        [524].S.BITS1.9   // 110-QUE-001-2 Sobrecarga
        [531].S.BITS1.9   // 110-ESC-002/3 Sobrecarga
        [184].S.BITS2.31   // 100-TOR-005 OUT MARCHA
        [283].S.BITS1.0   // 70-MIX-001-M Enable
        [283].S.BITS1.1   // 70-MIX-001-M Falla Resumen
        [283].S.BITS1.2   // 70-MIX-001-M Conf. Marcha
        [283].S.BITS1.26   // 70-MIX-001-M FLL
        [283].S.BITS1.27   // 70-MIX-001-M FV0
        [283].S.BITS1.28   // 70-MIX-001-M FATO
        [283].S.BITS1.30   // 70-MIX-001-M Falla Partida
        [283].S.BITS2.11   // ELE-060-00 Enc Ext
        [283].S.BITS2.20   // 70-MIX-001-M Reset Falla
        [283].S.BITS2.23   // 70-MIX-001-M Test
        [283].S.BITS2.27   // 70-MIX-001-M Cmd. Marcha
        [283].S.BITS2.30   // 70-MIX-001-M OUT MARCHA
        [283].S.BITS2.31   // ELE-060-00 Out
        [537].S.BITS1.9   // 110-ESC-004/3 Sobrecarga
        [187].S.BITS2.31   // 100-TOR-006 OUT MARCHA
        [276].S.BITS1.9   // 100-DOS-001-M08 Sobrecarga
        [284].S.BITS1.10   // 100-DOS-100-M12 Velocidad Cero
        [356].S.BITS1.9   // 110-CAN-004 Conf. Cerrado
        [284].S.BITS2.7   // BIF-061-00 Disable Codes
        [193].S.BITS2.31   // 100-TOR-007 OUT MARCHA
        [196].S.BITS2.31   // 100-TOR-008 OUT MARCHA
        [272].S.BITS1.8   // 100-DOS-001-M06 Atollo
        [285].S.BITS1.0   // 70-MIX-001-C Enable
        [285].S.BITS1.1   // 70-MIX-001-C Falla Resumen
        [285].S.BITS1.2   // 70-MIX-001-C Conf Pos Abrir
        [285].S.BITS1.4   // 70-MIX-001-C Conf Pos Cerrar
        [285].S.BITS1.29   // 70-MIX-001-C Falla Abrir
        [285].S.BITS1.30   // 70-MIX-001-C Falla Cerrar
        [285].S.BITS2.20   // 70-MIX-001-C Reset Falla
        [285].S.BITS2.23   // 70-MIX-001-C Test
        [285].S.BITS2.27   // 70-MIX-001-C Cmd. Open
        [285].S.BITS2.30   // 70-MIX-001-C OUT CLOSE
        [285].S.BITS2.31   // 70-MIX-001-C OUT OPEN
        [286].S.BITS1.0   // 70-TDC-012 Enable
        [286].S.BITS1.1   // 70-TDC-012 Falla Resumen
        [286].S.BITS1.2   // 70-TDC-012 Conf. Marcha
        [286].S.BITS1.3   // Conf Centro
        [286].S.BITS1.4   // 70-TDC-012 Cmd. Automatico
        [286].S.BITS1.8   // TOL-LISINA LL
        [286].S.BITS1.9   // TOL-LISINA LM
        [286].S.BITS1.10   // TOL-LISINA LH
        [286].S.BITS1.11   // C IZQUIERDA
        [286].S.BITS1.26   // 70-TDC-012 FLL
        [286].S.BITS1.27   // 70-TDC-012 FV0
        [286].S.BITS1.28   // 70-TDC-012 FATO
        [286].S.BITS1.30   // 70-TDC-012 Falla Partida
        [286].S.BITS2.11   // RED-062-00 Enc Ext
        [286].S.BITS2.20   // 70-TDC-012 Reset Falla
        [286].S.BITS2.23   // 70-TDC-012 Test
        [286].S.BITS2.25   // CMD IZQUIERDA
        [286].S.BITS2.26   // CDM CENTRO
        [286].S.BITS2.27   // 70-TDC-012 Cmd. Marcha
        [286].S.BITS2.29   // OUT IZQ
        [286].S.BITS2.30   // 70-TDC-012 OUT MARCHA
        [286].S.BITS2.31   // OUT DERECHA
        [287].S.BITS1.0   // 70-ELV-004 Enable
        [287].S.BITS1.1   // 70-ELV-004 Falla Resumen
        [287].S.BITS1.2   // 70-ELV-004 Conf. Marcha
        [287].S.BITS1.4   // 70-ELV-004 Cmd. Automatico
        [287].S.BITS1.26   // 70-ELV-004 FLL
        [287].S.BITS1.27   // 70-ELV-004 FV0
        [287].S.BITS1.28   // 70-ELV-004 FATO
        [287].S.BITS1.30   // 70-ELV-004 Falla Partida
        [287].S.BITS2.20   // 70-ELV-004 Reset Falla
        [287].S.BITS2.23   // 70-ELV-004 Test
        [287].S.BITS2.27   // 70-ELV-004 Cmd. Marcha
        [287].S.BITS2.30   // 70-ELV-004 OUT MARCHA
        [287].S.BITS2.31   // OUT DERECHA
        [288].S.BITS1.7   // TOLV-006 LLL
        [288].S.BITS1.8   // TOLV-006 LL
        [288].S.BITS1.9   // TOLV-006 LM
        [288].S.BITS1.10   // TOLV-006 LH
        [288].S.BITS1.26   // BOMB-LIQ4-B FLL
        [288].S.BITS1.27   // BOMB-LIQ4-B FV0
        [288].S.BITS1.28   // BOMB-LIQ4-B FATO
        [288].S.BITS2.27   // 100-DOS-001-C Cmd. Open
        [288].S.BITS2.30   // 100-DOS-001-C OUT CLOSE
        [540].S.BITS1.9   // 110-VEN-002/3 Sobrecarga
        [289].S.BITS1.2   // 100-TDP-003 Conf. Marcha
        [278].S.BITS1.9   // 100-DOS-001-M09 Sobrecarga
        [289].S.BITS1.29   // CV-MIX-001 Falla Abrir
        [544].S.BITS1.9   // 110-TOR-002/3 Sobrecarga
        [199].S.BITS2.31   // 100-TOR-009 OUT MARCHA
        [537].S.BITS1.8   // 110-ESC-004/3 Atollo
        [540].S.BITS1.8   // 110-VEN-002/3 Atollo
        [290].S.BITS1.0   // 80-TDC-001 Enable
        [290].S.BITS1.1   // 80-TDC-001 Falla Resumen
        [290].S.BITS1.2   // 80-TDC-001 Conf. Marcha
        [290].S.BITS1.4   // 80-TDC-001 Cmd. Automatico
        [290].S.BITS1.26   // 80-TDC-001 FLL
        [290].S.BITS1.27   // 80-TDC-001 FV0
        [290].S.BITS1.28   // 80-TDC-001 FATO
        [290].S.BITS1.29   // VAL-LIQ4-B Falla Abrir
        [290].S.BITS1.30   // 80-TDC-001 Falla Partida
        [290].S.BITS2.20   // 80-TDC-001 Reset Falla
        [290].S.BITS2.23   // 80-TDC-001 Test
        [290].S.BITS2.27   // 80-TDC-001 Cmd. Marcha
        [290].S.BITS2.30   // 80-TDC-001 OUT MARCHA
        [290].S.BITS2.31   // VAL-LIQ4-B OUT OPEN
        [291].S.BITS1.0   // DISP Enable
        [291].S.BITS1.1   // DISP Falla Resumen
        [291].S.BITS1.2   // DISP Conf Pos Abrir
        [291].S.BITS1.4   // DISP Conf Pos Cerrar
        [291].S.BITS1.7   // 80-TOL-001 LLL
        [291].S.BITS1.8   // 80-TOL-001 LL
        [291].S.BITS1.9   // 80-TOL-001 LM
        [291].S.BITS1.10   // 80-TOL-001 LH
        [291].S.BITS1.29   // DISP Falla Abrir
        [291].S.BITS1.30   // DISP Falla Cerrar
        [291].S.BITS2.20   // DISP Reset Falla
        [291].S.BITS2.23   // DISP Test
        [291].S.BITS2.27   // DISP Cmd. Open
        [291].S.BITS2.30   // DISP OUT CLOSE
        [291].S.BITS2.31   // DISP OUT OPEN
        [292].S.BITS1.0   // 100-TDP-004 Enable
        [292].S.BITS1.1   // 100-TDP-004 Falla Resumen
        [292].S.BITS1.2   // 100-TDP-004 Conf. Marcha
        [292].S.BITS1.4   // 100-TDP-004 Cmd. Automatico
        [292].S.BITS1.29   // 80-LMG-001-M1 Falla Abrir
        [292].S.BITS1.30   // 100-TDP-004 Falla Partida
        [292].S.BITS2.20   // 100-TDP-004 Reset Falla
        [292].S.BITS2.23   // 100-TDP-004 Test
        [292].S.BITS2.27   // 100-TDP-004 Cmd. Marcha
        [292].S.BITS2.30   // 100-TDP-004 OUT MARCHA
        [292].S.BITS2.31   // 100-TDP-004 OUT MARCHA
        [293].S.BITS1.0   // 100-ELV-002 Enable
        [293].S.BITS1.1   // 100-ELV-002 Falla Resumen
        [293].S.BITS1.4   // 100-ELV-002 Cmd. Automatico
        [293].S.BITS1.29   // 80-LMG-001-M2Falla Abrir
        [293].S.BITS1.30   // 100-ELV-002 Falla Partida
        [293].S.BITS2.20   // 100-ELV-002 Reset Falla
        [293].S.BITS2.23   // 100-ELV-002 Test
        [202].S.BITS2.31   // 100-TOR-010 OUT MARCHA
        [293].S.BITS2.30   // 100-ELV-002 OUT MARCHA
        [545].S.BITS1.9   // 110-TOR-003/3 Sobrecarga
        [294].S.BITS1.2   // 100-TDP-005 Conf. Marcha
        [294].S.BITS1.4   // 100-TDP-005 Cmd. Automatico
        [294].S.BITS1.30   // 100-TDP-005 Falla Partida
        [205].S.BITS2.31   // 100-TOR-036 OUT MARCHA
        [294].S.BITS2.27   // 100-TDP-005 Cmd. Marcha
        [294].S.BITS2.30   // 100-TDP-005 OUT MARCHA
        [294].S.BITS2.31   // 100-TDP-005 OUT MARCHA
        [295].S.BITS1.7   // 80-LMG-002-T LLL
        [295].S.BITS1.8   // 80-LMG-002-T LL
        [295].S.BITS1.9   // 80-LMG-002-T LM
        [295].S.BITS1.10   // 80-LMG-002-T LH
        [296].S.BITS1.7   // 80-TOL-002 LLL
        [297].S.BITS1.26   // 80-LRT-001 FLL
        [297].S.BITS1.27   // 80-LRT-001 FV0
        [297].S.BITS1.28   // 80-LRT-001 FATO
        [298].S.BITS1.0   // M1-COMP-401 Enable
        [298].S.BITS1.1   // M1-COMP-401 Falla Resumen
        [298].S.BITS1.2   // M1-COMP-401 Conf Pos Abrir
        [298].S.BITS1.4   // M1-COMP-401 Conf Pos Cerrar
        [298].S.BITS1.7   // 80-TOL-005 LLL
        [298].S.BITS1.8   // 80-TOL-005 LL
        [298].S.BITS1.9   // 80-TOL-005 LM
        [298].S.BITS1.10   // 80-TOL-005 LH
        [298].S.BITS1.29   // M1-COMP-401 Falla Abrir
        [298].S.BITS1.30   // M1-COMP-401 Falla Cerrar
        [298].S.BITS2.20   // M1-COMP-401 Reset Falla
        [298].S.BITS2.23   // M1-COMP-401 Test
        [298].S.BITS2.27   // M1-COMP-401 Cmd. Open
        [298].S.BITS2.30   // M1-COMP-401 OUT CLOSE
        [298].S.BITS2.31   // M1-COMP-401 OUT OPEN
        [546].S.BITS1.9   // 110-ELV-002/3 Sobrecarga
        [208].S.BITS2.31   // 100-TOR-012 OUT MARCHA
        [280].S.BITS1.9   // 100-DOS-100-M10 Sobrecarga
        [357].S.BITS1.9   // 110-CAN-005 Conf. Cerrado
        [211].S.BITS2.31   // 100-TOR-013 OUT MARCHA
        [214].S.BITS2.31   // 100-TOR-014 OUT MARCHA
        [274].S.BITS1.8   // 100-DOS-001-M07 Atollo
        [301].S.BITS1.7   // 80-TOL-003 LLL
        [548].S.BITS1.9   // 110-TOR-004/3 Sobrecarga
        [217].S.BITS2.31   // 100-TOR-015 OUT MARCHA
        [282].S.BITS1.9   // 100-DOS-100-M11 Sobrecarga
        [358].S.BITS1.9   // 8-ENF-730 LM
        [218].S.BITS2.31   // 100-TOR-038 OUT MARCHA
        [220].S.BITS2.31   // 100-TOR-011 OUT MARCHA
        [276].S.BITS1.8   // 100-DOS-001-M08 Atollo
        [303].S.BITS1.0   // XY-6170 Enable
        [303].S.BITS1.1   // XY-6170 Falla Resumen
        [303].S.BITS1.2   // XY-6170 Conf. Marcha
        [303].S.BITS1.4   // XY-6170 Cmd. Automatico
        [303].S.BITS1.29   // 80-CAN-001 Falla Abrir
        [303].S.BITS1.30   // XY-6170 Falla Partida
        [303].S.BITS2.20   // XY-6170 Reset Falla
        [303].S.BITS2.23   // XY-6170 Test
        [303].S.BITS2.27   // XY-6170 Cmd. Marcha
        [303].S.BITS2.30   // XY-6170 OUT MARCHA
        [303].S.BITS2.31   // XY-6170 OUT MARCHA
        [551].S.BITS1.9   // 110-TDC-003/1 Sobrecarga
        [304].S.BITS1.2   // 100-BCE-005 Conf. Marcha
        [284].S.BITS1.9   // 100-DOS-100-M12 Sobrecarga
        [304].S.BITS1.29   // 80-CAN-002 Falla Abrir
        [552].S.BITS1.9   // 110-TDC-004/1 Sobrecarga
        [223].S.BITS2.31   // 100-TOR-035 OUT MARCHA
        [544].S.BITS1.8   // 110-TOR-002/3 Atollo
        [545].S.BITS1.8   // 110-TOR-003/3 Atollo
        [305].S.BITS1.0   // XY-6171 Enable
        [305].S.BITS1.1   // XY-6171 Falla Resumen
        [305].S.BITS1.2   // XY-6171 Conf. Marcha
        [305].S.BITS1.4   // XY-6171 Cmd. Automatico
        [305].S.BITS1.26   // XY-6171 FLL
        [305].S.BITS1.27   // XY-6171 FV0
        [305].S.BITS1.28   // XY-6171 FATO
        [305].S.BITS1.29   // 80-CAN-003 Falla Abrir
        [305].S.BITS1.30   // XY-6171 Falla Partida
        [305].S.BITS2.20   // XY-6171 Reset Falla
        [305].S.BITS2.23   // XY-6171 Test
        [305].S.BITS2.27   // XY-6171 Cmd. Marcha
        [305].S.BITS2.30   // XY-6171 OUT MARCHA
        [305].S.BITS2.31   // XY-6171 OUT MARCHA
        [306].S.BITS1.29   // 80-CAN-004 Falla Abrir
        [306].S.BITS2.31   // XY-6121 OUT MARCHA
        [307].S.BITS1.0   // 80-TDC-005 Enable
        [307].S.BITS1.1   // 80-TDC-005 Falla Resumen
        [307].S.BITS1.2   // 80-TDC-005 Conf. Marcha
        [307].S.BITS1.4   // 80-TDC-005 Cmd. Automatico
        [307].S.BITS1.26   // 80-TDC-005 FLL
        [307].S.BITS1.27   // 80-TDC-005 FV0
        [307].S.BITS1.28   // 80-TDC-005 FATO
        [307].S.BITS1.30   // 80-TDC-005 Falla Partida
        [307].S.BITS2.20   // 80-TDC-005 Reset Falla
        [307].S.BITS2.23   // 80-TDC-005 Test
        [307].S.BITS2.27   // 80-TDC-005 Cmd. Marcha
        [307].S.BITS2.30   // 80-TDC-005 OUT MARCHA
        [554].S.BITS1.9   // 110-ELV-001/1 Sobrecarga
        [234].S.BITS2.27   // 100-CAN-023 Cmd. Open
        [314].S.BITS1.9   // 100-VEN-ACORG-1 Sobrecarga
        [308].S.BITS1.7   // 80-TOL-RED1 LLL
        [308].S.BITS1.10   // 100-BCE-002 Velocidad Cero
        [557].S.BITS1.9   // 120-XY-8127 Conf. Cerrado
        [234].S.BITS2.30   // 100-CAN-023 OUT CLOSE
        [236].S.BITS2.27   // 100-CAN-025 Cmd. Open
        [278].S.BITS1.8   // 100-DOS-001-M09 Atollo
        [310].S.BITS1.7   // 80-TOL-004/5 LLL
        [310].S.BITS1.8   // 80-TOL-004/5 LL
        [310].S.BITS1.9   // 80-TOL-004/5 LM
        [310].S.BITS1.10   // 80-TOL-004/5 LH
        [311].S.BITS1.0   // 8-PLT-622 Enable
        [311].S.BITS1.1   // 8-PLT-622 Falla Resumen
        [311].S.BITS1.2   // 8-PLT-622 Conf. Marcha
        [311].S.BITS1.4   // 8-PLT-622 Cmd. Automatico
        [311].S.BITS1.26   // 8-PLT-622 FLL
        [311].S.BITS1.27   // 8-PLT-622 FV0
        [311].S.BITS1.28   // 8-PLT-622 FATO
        [311].S.BITS1.30   // 8-PLT-622 Falla Partida
        [311].S.BITS2.20   // 8-PLT-622 Reset Falla
        [311].S.BITS2.23   // 8-PLT-622 Test
        [311].S.BITS2.27   // 8-PLT-622 Cmd. Marcha
        [311].S.BITS2.30   // 8-PLT-622 OUT MARCHA
        [312].S.BITS1.0   // 8-BIF-624 Enable
        [312].S.BITS1.1   // 8-BIF-624 Falla Resumen
        [312].S.BITS1.26   // 100-BCE-001 FLL
        [312].S.BITS1.27   // 100-BCE-001 FV0
        [312].S.BITS1.28   // 100-BCE-001 FATO
        [312].S.BITS2.20   // 8-BIF-624 Reset Falla
        [312].S.BITS2.23   // 8-BIF-624 Test
        [313].S.BITS1.0   // XY-6102 Enable
        [313].S.BITS1.1   // XY-6102 Falla Resumen
        [313].S.BITS1.2   // XY-6102 Conf. Marcha
        [313].S.BITS1.3   // M1-TRI-095 Conf. Pos. Centro
        [313].S.BITS1.4   // XY-6102 Cmd. Automatico
        [313].S.BITS1.29   // M1-TRI-095 Falla Pos. Centro
        [313].S.BITS1.30   // XY-6102 Falla Partida
        [313].S.BITS2.20   // XY-6102 Reset Falla
        [313].S.BITS2.23   // XY-6102 Test
        [313].S.BITS2.26   // M1-TRI-095 Cmd. Pos . Centro
        [313].S.BITS2.27   // XY-6102 Cmd. Marcha
        [313].S.BITS2.30   // XY-6102 OUT MARCHA
        [313].S.BITS2.31   // XY-6102 OUT MARCHA
        [332].S.BITS1.8   // 110-FIL-001 Atollo
        [315].S.BITS1.9   // 100-VEN-ACORG-2 Sobrecarga
        [559].S.BITS1.9   // 120-CAN-001 Conf. Cerrado
        [152].S.BITS1.10   // 100-TDC-005 Velocidad Cero
        [182].S.BITS1.8   // 7-DOS-1170-05 LL
        [84].S.BITS1.10   // 90-MRO-003-B Velocidad Cero
        [567].S.BITS1.9   // 120-XY-8128 Conf. Cerrado
        [187].S.BITS1.8   // 100-TOR-006 Atollo
        [569].S.BITS1.9   // 120-CAN-003 Conf. Cerrado
        [555].S.BITS1.9   // 120-TDC-001/1 Sobrecarga
        [334].S.BITS1.8   // 110-FIL-002 Atollo
        [353].S.BITS1.10   // 110-CAN-001 Conf. Abierto
        [577].S.BITS1.9   // 120-XY-8129 Conf. Cerrado
        [157].S.BITS1.10   // 100-TDC-006 Velocidad Cero
        [193].S.BITS1.8   // 100-TOR-007 Atollo
        [112].S.BITS1.10   // 100-FIL-001 Velocidad Cero
        [582].S.BITS1.9   // 120-CAN-007 Conf. Cerrado
        [196].S.BITS1.8   // 7-DOS-1170-12 LL
        [583].S.BITS1.9   // 120-CAN-008 Conf. Cerrado
        [561].S.BITS1.9   // 110-TDC-003/2 Sobrecarga
        [336].S.BITS1.8   // 110-FIL-003 Atollo
        [354].S.BITS1.10   // 110-CAN-002 Conf. Abierto
        [584].S.BITS1.9   // 120-CAN-009 Conf. Cerrado
        [168].S.BITS1.10   // 100-FIL-002 Velocidad Cero
        [199].S.BITS1.8   // 100-TOR-009 Atollo
        [113].S.BITS1.10   // 7-BIN-1112 LH
        [585].S.BITS1.9   // 120-CAN-010 Conf. Cerrado
